RoboDK station: kr30 cnc 070119 is there hope.rdk

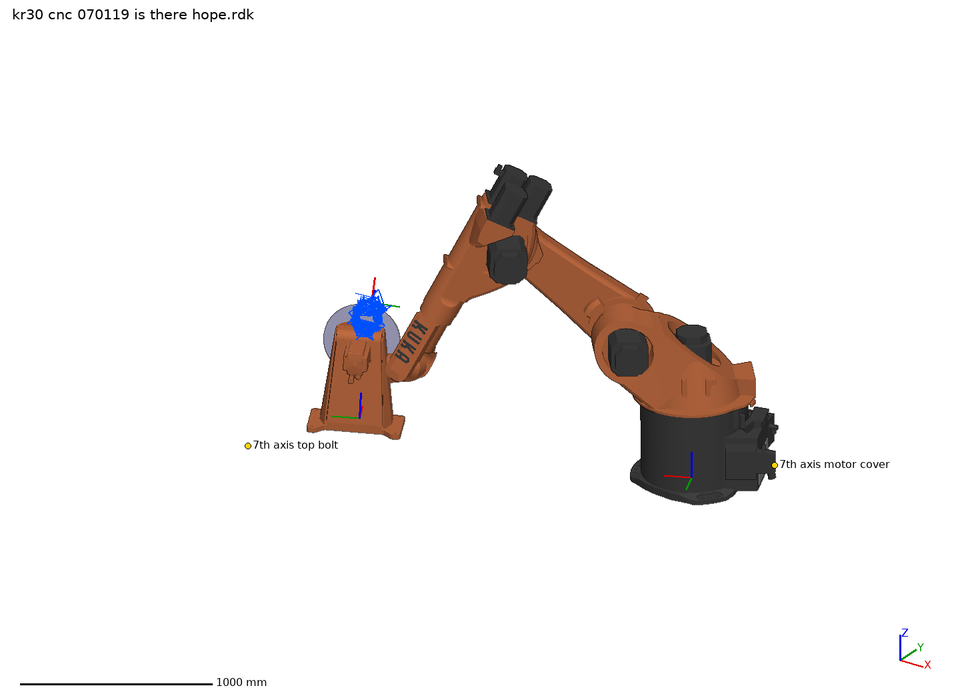
[picture v0: the station drawn from its stored meshes, robots at their saved joint values, targets as dots, program paths as lines]
Station kr30 cnc 070119 is there hope. Poses are relative to the parent item; angles as X-Y-Z fixed-axis rotations.
  - frame KUKA KR 30 HA Base at (1535.48, 628.29, -1072.61) mm, rotated rx 0 ry 0 rz -156.31 deg
    - robot KUKA KR 30 HA: 6 axes, payload 30 kg, reach 2033 mm, repeatability 0.05 mm, weight 665 kg
        modified DH rows (alpha deg, a mm, theta deg, d mm): 0, 0, 0, 815; -90, 350, 0, 0; 0, 850, -90, 0; -90, 145, 0, 820; 90, 0, 0, 0; -90, 0, 180, 170
        joint limits [-185, -135, -120, -350, -119, -350] to [185, 35, 158, 350, 119, 350]; home [0, -90, 90, 0, 0, 0]; saved at [-17.375, -41.925, 104.176, 143.001, 49.162, -26.712]
      - tool 1/2" End Mill TCP, TCP at (337.71, -2.2, 160.57) mm, rotated rx 0 ry 90 rz 0 deg, size 415.8 x 102 x 153.6 mm
    - target 7th axis top bolt (joint target) at (1966.13, 1947.63, 927.26) mm, rotated rx -179.2 ry 6.72 rz -171.11 deg; joints [-17.018, -71.525, 110.046, 168.711, 45.865, -170.331, 883.939] of KUKA KR 30 HA
    - target 7th axis motor cover (joint target) at (-417, -111.35, 57.2) mm, rotated rx -135.46 ry -1.69 rz -48.75 deg; joints [-33.388, -54.543, 96.086, 147.711, 45.276, -113.831, 883.939] of KUKA KR 30 HA
  - frame KUKA KP1 MD250 Base at (172.34, -439.05, -684.5) mm, rotated rx 2 ry 0.52 rz 120.23 deg
    - robot KUKA KP1 MD250: 1 axes, payload 250 kg
        modified DH rows (alpha deg, a mm, theta deg, d mm): 0, 0, 0, 0
        base shift (70, 10, 428) mm, rotated rx 0 ry 90 rz -2 deg
        joint limits [-3600] to [3600]; home [0]; saved at [-175]
      - frame Frame 2 at (0, 0, 440) mm
  - machining project Machining Settings: C:/Users/liqui/OneDrive/Desktop/suffering.apt | rotz(5) | rotz(0)
  - program Machining (7499 instructions, listed below)
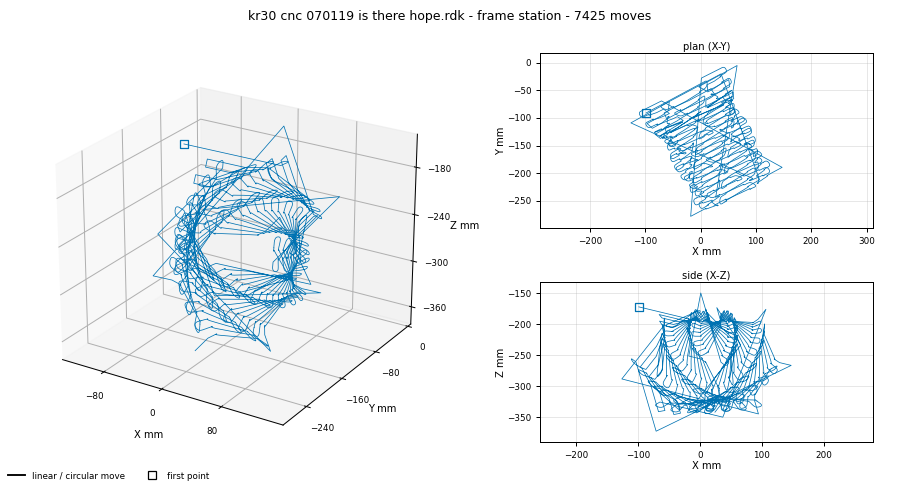
[picture p0: tool path of kr30 cnc 070119 is there hope.rdk in frame station, 7425 of 7425 moves have a stored position in this frame; points joined in program order, loops and branches not executed]

--- program Machining (robot KUKA KR 30 HA) ---
  Smooth(1)
  Set Ref.: Frame 2
  Set Tool: 1/2" End Mill TCP
  Show 1/2" End Mill TCP
  Print: /'1001'
  Print: /''
  Print: /'Flow1'
  Set speed (1000.0 mm/s)
  Set speed (1000.0 mm/s)
  MoveJ 1 to (79.06, -86.72, -80.22) mm, rotated rx 42.04 ry 15.1 rz 65.25 deg; joints [-11.881, -44.556, 105.513, 149.142, 46.632, -28.661, -175]
  MoveL 2 to (79.06, -86.72, -80.22) mm, rotated rx 42.04 ry 15.1 rz 65.25 deg; joints [-11.881, -44.556, 105.513, 149.142, 46.632, -28.661, -175]
  MoveL 3 to (79.06, -86.72, -80.22) mm, rotated rx 42.04 ry 15.1 rz 65.25 deg; joints [-11.881, -44.556, 105.513, 149.142, 46.632, -28.661, -175]
  Set speed (1000.0 mm/s)
  MoveL 4 to (75.15, -42.01, -80.22) mm, rotated rx 42.04 ry 15.1 rz 65.25 deg; joints [-12.109, -45.867, 109.411, 150.046, 48.916, -30.305, -175]
  Set speed (100.0 mm/s)
  MoveL 5 to (68.81, 30.47, -80.22) mm, rotated rx 42.04 ry 15.1 rz 65.25 deg; joints [-12.508, -47.756, 115.477, 151.236, 52.637, -32.762, -175]
  MoveL 6 to (69.1, 30.91, -80.22) mm, rotated rx 42.04 ry 15.1 rz 65.25 deg; joints [-12.511, -47.788, 115.518, 151.237, 52.647, -32.767, -175]
  MoveL 7 to (69.4, 31.48, -80.12) mm, rotated rx 42.04 ry 15.1 rz 65.25 deg; joints [-12.51, -47.824, 115.571, 151.244, 52.661, -32.777, -175]
  MoveL 8 to (69.7, 31.99, -80.06) mm, rotated rx 42.04 ry 15.1 rz 65.25 deg; joints [-12.511, -47.858, 115.619, 151.248, 52.674, -32.786, -175]
  MoveL 9 to (70, 32.47, -80.04) mm, rotated rx 42.04 ry 15.1 rz 65.25 deg; joints [-12.513, -47.891, 115.664, 151.25, 52.685, -32.792, -175]
  MoveL 10 to (72, 35.54, -80.04) mm, rotated rx 42.04 ry 15.1 rz 65.25 deg; joints [-12.532, -48.109, 115.952, 151.254, 52.75, -32.827, -175]
  MoveL 11 to (72.84, 36.72, -80.13) mm, rotated rx 42.04 ry 15.1 rz 65.25 deg; joints [-12.542, -48.197, 116.063, 151.249, 52.771, -32.836, -175]
  MoveL 12 to (73.64, 37.61, -80.4) mm, rotated rx 42.04 ry 15.1 rz 65.25 deg; joints [-12.559, -48.272, 116.146, 151.233, 52.781, -32.834, -175]
  MoveL 13 to (74.38, 38.19, -80.84) mm, rotated rx 42.04 ry 15.1 rz 65.25 deg; joints [-12.581, -48.334, 116.201, 151.204, 52.779, -32.82, -175]
  MoveL 14 to (74.73, 38.37, -81.13) mm, rotated rx 42.04 ry 15.1 rz 65.25 deg; joints [-12.594, -48.361, 116.218, 151.185, 52.774, -32.809, -175]
  MoveL 15 to (75.07, 38.48, -81.46) mm, rotated rx 42.04 ry 15.1 rz 65.25 deg; joints [-12.609, -48.384, 116.229, 151.163, 52.765, -32.795, -175]
  MoveL 16 to (75.72, 38.47, -82.26) mm, rotated rx 42.04 ry 15.1 rz 65.25 deg; joints [-12.642, -48.421, 116.229, 151.11, 52.739, -32.759, -175]
  MoveL 17 to (76.31, 38.17, -83.24) mm, rotated rx 42.04 ry 15.1 rz 65.25 deg; joints [-12.682, -48.445, 116.202, 151.045, 52.701, -32.712, -175]
  MoveL 18 to (77.36, 36.66, -85.72) mm, rotated rx 42.04 ry 15.1 rz 65.25 deg; joints [-12.777, -48.455, 116.064, 150.878, 52.589, -32.582, -175]
  MoveL 19 to (77.93, 34.52, -88.21) mm, rotated rx 42.04 ry 15.1 rz 65.25 deg; joints [-12.867, -48.415, 115.865, 150.712, 52.467, -32.446, -175]
  MoveL 20 to (77.76, 32.29, -89.98) mm, rotated rx 42.04 ry 15.1 rz 65.25 deg; joints [-12.927, -48.329, 115.655, 150.594, 52.371, -32.344, -175]
  MoveL 21 to (77.39, 31.15, -90.6) mm, rotated rx 42.04 ry 15.1 rz 65.25 deg; joints [-12.946, -48.269, 115.547, 150.554, 52.332, -32.306, -175]
  MoveL 22 to (76.84, 29.98, -91.05) mm, rotated rx 42.04 ry 15.1 rz 65.25 deg; joints [-12.957, -48.197, 115.435, 150.526, 52.3, -32.277, -175]
  MoveL 23 to (75.19, 27.58, -91.4) mm, rotated rx 42.04 ry 15.1 rz 65.25 deg; joints [-12.956, -48.019, 115.205, 150.507, 52.254, -32.244, -175]
  MoveL 24 to (73.18, 25.16, -91.41) mm, rotated rx 42.04 ry 15.1 rz 65.25 deg; joints [-12.941, -47.82, 114.97, 150.511, 52.22, -32.229, -175]
  MoveL 25 to (72.87, 24.77, -91.43) mm, rotated rx 42.04 ry 15.1 rz 65.25 deg; joints [-12.94, -47.789, 114.933, 150.51, 52.214, -32.225, -175]
  MoveL 26 to (72.6, 24.4, -91.47) mm, rotated rx 42.04 ry 15.1 rz 65.25 deg; joints [-12.939, -47.761, 114.897, 150.508, 52.208, -32.221, -175]
  MoveL 27 to (72.37, 24.06, -91.53) mm, rotated rx 42.04 ry 15.1 rz 65.25 deg; joints [-12.939, -47.735, 114.864, 150.505, 52.201, -32.216, -175]
  MoveL 28 to (72.11, 23.7, -91.58) mm, rotated rx 42.04 ry 15.1 rz 65.25 deg; joints [-12.939, -47.708, 114.829, 150.502, 52.194, -32.211, -175]
  MoveL 29 to (71.77, 23.27, -91.6) mm, rotated rx 42.04 ry 15.1 rz 65.25 deg; joints [-12.937, -47.674, 114.787, 150.501, 52.187, -32.207, -175]
  MoveL 30 to (71.37, 22.75, -91.64) mm, rotated rx 42.04 ry 15.1 rz 65.25 deg; joints [-12.936, -47.633, 114.737, 150.5, 52.179, -32.202, -175]
  MoveL 31 to (71.04, 22.3, -91.7) mm, rotated rx 42.04 ry 15.1 rz 65.25 deg; joints [-12.935, -47.599, 114.693, 150.497, 52.171, -32.197, -175]
  MoveL 32 to (70.79, 21.93, -91.77) mm, rotated rx 42.04 ry 15.1 rz 65.25 deg; joints [-12.936, -47.571, 114.657, 150.493, 52.163, -32.191, -175]
  MoveL 33 to (70.54, 21.58, -91.82) mm, rotated rx 42.04 ry 15.1 rz 65.25 deg; joints [-12.936, -47.545, 114.623, 150.49, 52.157, -32.186, -175]
  MoveL 34 to (70.24, 21.2, -91.84) mm, rotated rx 42.04 ry 15.1 rz 65.25 deg; joints [-12.934, -47.515, 114.586, 150.489, 52.151, -32.183, -175]
  MoveL 35 to (69.91, 20.8, -91.84) mm, rotated rx 42.04 ry 15.1 rz 65.25 deg; joints [-12.932, -47.482, 114.547, 150.49, 52.145, -32.18, -175]
  MoveL 36 to (69.56, 20.38, -91.85) mm, rotated rx 42.04 ry 15.1 rz 65.25 deg; joints [-12.929, -47.448, 114.506, 150.491, 52.139, -32.177, -175]
  MoveL 37 to (69.21, 19.93, -91.86) mm, rotated rx 42.04 ry 15.1 rz 65.25 deg; joints [-12.927, -47.412, 114.463, 150.49, 52.131, -32.173, -175]
  MoveL 38 to (68.81, 19.4, -91.89) mm, rotated rx 42.04 ry 15.1 rz 65.25 deg; joints [-12.925, -47.371, 114.412, 150.489, 52.122, -32.168, -175]
  MoveL 39 to (68.49, 18.91, -91.96) mm, rotated rx 42.04 ry 15.1 rz 65.25 deg; joints [-12.924, -47.335, 114.364, 150.485, 52.112, -32.16, -175]
  MoveL 40 to (68.26, 18.52, -92.06) mm, rotated rx 42.04 ry 15.1 rz 65.25 deg; joints [-12.926, -47.309, 114.326, 150.478, 52.102, -32.153, -175]
  MoveL 41 to (68.25, 18.52, -92.3) mm, rotated rx 42.04 ry 15.1 rz 65.25 deg; joints [-12.936, -47.307, 114.324, 150.466, 52.103, -32.148, -175]
  MoveL 42 to (68.39, 18.89, -92.65) mm, rotated rx 42.04 ry 15.1 rz 65.25 deg; joints [-12.953, -47.325, 114.353, 150.45, 52.115, -32.147, -175]
  MoveL 43 to (69.21, 19.13, -93.61) mm, rotated rx 42.04 ry 15.1 rz 65.25 deg; joints [-12.994, -47.379, 114.374, 150.389, 52.095, -32.109, -175]
  MoveL 44 to (68.99, 17.01, -93.61) mm, rotated rx 42.04 ry 15.1 rz 65.25 deg; joints [-12.981, -47.301, 114.192, 150.365, 52.003, -32.05, -175]
  MoveL 45 to (68.79, 14.72, -93.74) mm, rotated rx 42.04 ry 15.1 rz 65.25 deg; joints [-12.972, -47.219, 113.996, 150.33, 51.902, -31.982, -175]
  MoveL 46 to (68.58, 12.55, -93.8) mm, rotated rx 42.04 ry 15.1 rz 65.25 deg; joints [-12.961, -47.139, 113.809, 150.302, 51.807, -31.919, -175]
  MoveL 47 to (68.38, 10.44, -93.93) mm, rotated rx 42.04 ry 15.1 rz 65.25 deg; joints [-12.954, -47.062, 113.627, 150.27, 51.714, -31.856, -175]
  MoveL 48 to (68.18, 8.3, -94.09) mm, rotated rx 42.04 ry 15.1 rz 65.25 deg; joints [-12.947, -46.984, 113.442, 150.236, 51.62, -31.791, -175]
  MoveL 49 to (67.98, 6.19, -94.21) mm, rotated rx 42.04 ry 15.1 rz 65.25 deg; joints [-12.94, -46.906, 113.259, 150.203, 51.527, -31.728, -175]
  MoveL 50 to (67.78, 4.06, -94.42) mm, rotated rx 42.04 ry 15.1 rz 65.25 deg; joints [-12.935, -46.827, 113.073, 150.166, 51.433, -31.662, -175]
  MoveL 51 to (67.57, 1.94, -94.54) mm, rotated rx 42.04 ry 15.1 rz 65.25 deg; joints [-12.927, -46.748, 112.889, 150.134, 51.34, -31.599, -175]
  MoveL 52 to (67.36, -0.19, -94.59) mm, rotated rx 42.04 ry 15.1 rz 65.25 deg; joints [-12.917, -46.669, 112.704, 150.105, 51.247, -31.536, -175]
  MoveL 53 to (67.14, -2.34, -94.74) mm, rotated rx 42.04 ry 15.1 rz 65.25 deg; joints [-12.91, -46.588, 112.517, 150.07, 51.153, -31.471, -175]
  MoveL 54 to (66.92, -4.55, -94.92) mm, rotated rx 42.04 ry 15.1 rz 65.25 deg; joints [-12.904, -46.505, 112.323, 150.033, 51.056, -31.403, -175]
  MoveL 55 to (66.69, -6.77, -95.1) mm, rotated rx 42.04 ry 15.1 rz 65.25 deg; joints [-12.898, -46.421, 112.128, 149.995, 50.959, -31.335, -175]
  MoveL 56 to (66.49, -8.63, -95.34) mm, rotated rx 42.04 ry 15.1 rz 65.25 deg; joints [-12.896, -46.349, 111.963, 149.959, 50.878, -31.275, -175]
  MoveL 57 to (66.21, -11.29, -95.45) mm, rotated rx 42.04 ry 15.1 rz 65.25 deg; joints [-12.885, -46.248, 111.731, 149.919, 50.762, -31.196, -175]
  Set speed (1000.0 mm/s)
  MoveL 58 to (70.16, -56.42, -95.45) mm, rotated rx 42.04 ry 15.1 rz 65.25 deg; joints [-12.627, -45.013, 107.885, 149.106, 48.456, -29.584, -175]
  Set speed (1000.0 mm/s)
  MoveL 59 to (64.44, -56.92, -107.33) mm, rotated rx 42.04 ry 15.1 rz 65.25 deg; joints [-13.086, -44.596, 107.594, 148.598, 48.671, -29.432, -175]
  Set speed (100.0 mm/s)
  MoveL 60 to (61.94, -28.34, -107.33) mm, rotated rx 42.04 ry 15.1 rz 65.25 deg; joints [-13.255, -45.385, 110.042, 149.126, 50.129, -30.478, -175]
  MoveL 61 to (62.35, -26.67, -107.08) mm, rotated rx 42.04 ry 15.1 rz 65.25 deg; joints [-13.256, -45.465, 110.196, 149.157, 50.193, -30.527, -175]
  MoveL 62 to (62.8, -24.7, -107.02) mm, rotated rx 42.04 ry 15.1 rz 65.25 deg; joints [-13.266, -45.555, 110.375, 149.183, 50.271, -30.581, -175]
  MoveL 63 to (63.26, -22.7, -106.87) mm, rotated rx 42.04 ry 15.1 rz 65.25 deg; joints [-13.272, -45.648, 110.556, 149.213, 50.349, -30.637, -175]
  MoveL 64 to (63.83, -20.3, -106.74) mm, rotated rx 42.04 ry 15.1 rz 65.25 deg; joints [-13.282, -45.759, 110.773, 149.246, 50.442, -30.703, -175]
  MoveL 65 to (64.3, -18.22, -106.74) mm, rotated rx 42.04 ry 15.1 rz 65.25 deg; joints [-13.295, -45.854, 110.96, 149.269, 50.524, -30.758, -175]
  MoveL 66 to (64.81, -15.92, -106.58) mm, rotated rx 42.04 ry 15.1 rz 65.25 deg; joints [-13.303, -45.959, 111.167, 149.303, 50.614, -30.822, -175]
  MoveL 67 to (65.26, -13.98, -106.39) mm, rotated rx 42.04 ry 15.1 rz 65.25 deg; joints [-13.307, -46.048, 111.343, 149.333, 50.689, -30.877, -175]
  MoveL 68 to (65.72, -11.98, -106.3) mm, rotated rx 42.04 ry 15.1 rz 65.25 deg; joints [-13.316, -46.139, 111.523, 149.359, 50.767, -30.931, -175]
  MoveL 69 to (66.18, -9.9, -106.08) mm, rotated rx 42.04 ry 15.1 rz 65.25 deg; joints [-13.321, -46.234, 111.711, 149.393, 50.848, -30.99, -175]
  MoveL 70 to (66.64, -7.83, -105.93) mm, rotated rx 42.04 ry 15.1 rz 65.25 deg; joints [-13.327, -46.328, 111.896, 149.423, 50.928, -31.047, -175]
  MoveL 71 to (67.1, -5.77, -105.82) mm, rotated rx 42.04 ry 15.1 rz 65.25 deg; joints [-13.336, -46.421, 112.081, 149.45, 51.009, -31.103, -175]
  MoveL 72 to (67.55, -3.68, -105.65) mm, rotated rx 42.04 ry 15.1 rz 65.25 deg; joints [-13.342, -46.515, 112.268, 149.481, 51.091, -31.161, -175]
  MoveL 73 to (68, -1.6, -105.51) mm, rotated rx 42.04 ry 15.1 rz 65.25 deg; joints [-13.35, -46.608, 112.454, 149.51, 51.172, -31.218, -175]
  MoveL 74 to (68.47, 0.52, -105.44) mm, rotated rx 42.04 ry 15.1 rz 65.25 deg; joints [-13.361, -46.703, 112.642, 149.535, 51.255, -31.274, -175]
  MoveL 75 to (68.91, 2.61, -105.23) mm, rotated rx 42.04 ry 15.1 rz 65.25 deg; joints [-13.365, -46.796, 112.829, 149.567, 51.337, -31.333, -175]
  MoveL 76 to (69.35, 4.68, -105.11) mm, rotated rx 42.04 ry 15.1 rz 65.25 deg; joints [-13.374, -46.888, 113.013, 149.595, 51.418, -31.389, -175]
  MoveL 77 to (69.81, 6.8, -104.99) mm, rotated rx 42.04 ry 15.1 rz 65.25 deg; joints [-13.382, -46.982, 113.201, 149.622, 51.5, -31.446, -175]
  MoveL 78 to (70.05, 8.56, -104.78) mm, rotated rx 42.04 ry 15.1 rz 65.25 deg; joints [-13.385, -47.052, 113.356, 149.653, 51.574, -31.499, -175]
  MoveL 79 to (70.11, 10.03, -104.43) mm, rotated rx 42.04 ry 15.1 rz 65.25 deg; joints [-13.38, -47.103, 113.485, 149.691, 51.641, -31.552, -175]
  MoveL 80 to (69.98, 11.23, -103.9) mm, rotated rx 42.04 ry 15.1 rz 65.25 deg; joints [-13.366, -47.134, 113.591, 149.737, 51.702, -31.606, -175]
  MoveL 81 to (69.2, 9.9, -103.04) mm, rotated rx 42.04 ry 15.1 rz 65.25 deg; joints [-13.322, -47.05, 113.478, 149.777, 51.668, -31.607, -175]
  MoveL 82 to (69.54, 10.63, -103.04) mm, rotated rx 42.04 ry 15.1 rz 65.25 deg; joints [-13.327, -47.093, 113.544, 149.781, 51.69, -31.62, -175]
  MoveL 83 to (69.9, 11.23, -103.04) mm, rotated rx 42.04 ry 15.1 rz 65.25 deg; joints [-13.331, -47.134, 113.601, 149.783, 51.705, -31.628, -175]
  MoveL 84 to (70.3, 11.73, -103.04) mm, rotated rx 42.04 ry 15.1 rz 65.25 deg; joints [-13.334, -47.174, 113.649, 149.782, 51.712, -31.632, -175]
  MoveL 85 to (70.75, 12.22, -103.02) mm, rotated rx 42.04 ry 15.1 rz 65.25 deg; joints [-13.337, -47.217, 113.699, 149.782, 51.718, -31.635, -175]
  MoveL 86 to (71.28, 12.77, -102.98) mm, rotated rx 42.04 ry 15.1 rz 65.25 deg; joints [-13.339, -47.267, 113.754, 149.781, 51.723, -31.637, -175]
  MoveL 87 to (72.8, 14.21, -102.98) mm, rotated rx 42.04 ry 15.1 rz 65.25 deg; joints [-13.348, -47.405, 113.899, 149.773, 51.731, -31.638, -175]
  MoveL 88 to (73.12, 14.53, -102.96) mm, rotated rx 42.04 ry 15.1 rz 65.25 deg; joints [-13.35, -47.435, 113.931, 149.772, 51.734, -31.639, -175]
  MoveL 89 to (73.88, 15.25, -102.96) mm, rotated rx 42.04 ry 15.1 rz 65.25 deg; joints [-13.355, -47.504, 114.004, 149.768, 51.738, -31.639, -175]
  MoveL 90 to (74.24, 15.6, -102.96) mm, rotated rx 42.04 ry 15.1 rz 65.25 deg; joints [-13.357, -47.537, 114.039, 149.766, 51.74, -31.639, -175]
  MoveL 91 to (74.59, 15.94, -102.94) mm, rotated rx 42.04 ry 15.1 rz 65.25 deg; joints [-13.358, -47.569, 114.074, 149.765, 51.742, -31.64, -175]
  MoveL 92 to (74.92, 16.29, -102.91) mm, rotated rx 42.04 ry 15.1 rz 65.25 deg; joints [-13.359, -47.601, 114.109, 149.765, 51.745, -31.642, -175]
  MoveL 93 to (75.21, 16.61, -102.85) mm, rotated rx 42.04 ry 15.1 rz 65.25 deg; joints [-13.359, -47.629, 114.141, 149.767, 51.749, -31.645, -175]
  MoveL 94 to (75.53, 16.95, -102.81) mm, rotated rx 42.04 ry 15.1 rz 65.25 deg; joints [-13.36, -47.66, 114.176, 149.768, 51.752, -31.647, -175]
  MoveL 95 to (75.88, 17.3, -102.79) mm, rotated rx 42.04 ry 15.1 rz 65.25 deg; joints [-13.361, -47.693, 114.211, 149.767, 51.755, -31.647, -175]
  MoveL 96 to (76.25, 17.66, -102.78) mm, rotated rx 42.04 ry 15.1 rz 65.25 deg; joints [-13.363, -47.726, 114.246, 149.765, 51.757, -31.648, -175]
  MoveL 97 to (76.6, 18.01, -102.77) mm, rotated rx 42.04 ry 15.1 rz 65.25 deg; joints [-13.365, -47.759, 114.281, 149.764, 51.759, -31.649, -175]
  MoveL 98 to (76.92, 18.35, -102.73) mm, rotated rx 42.04 ry 15.1 rz 65.25 deg; joints [-13.366, -47.79, 114.316, 149.765, 51.763, -31.651, -175]
  MoveL 99 to (77.21, 18.68, -102.67) mm, rotated rx 42.04 ry 15.1 rz 65.25 deg; joints [-13.366, -47.818, 114.349, 149.767, 51.767, -31.654, -175]
  MoveL 100 to (77.51, 19.03, -102.62) mm, rotated rx 42.04 ry 15.1 rz 65.25 deg; joints [-13.366, -47.847, 114.383, 149.768, 51.771, -31.657, -175]
  MoveL 101 to (78.5, 20.06, -102.54) mm, rotated rx 42.04 ry 15.1 rz 65.25 deg; joints [-13.369, -47.942, 114.487, 149.768, 51.78, -31.661, -175]
  MoveL 102 to (79.42, 20.81, -102.66) mm, rotated rx 42.04 ry 15.1 rz 65.25 deg; joints [-13.38, -48.021, 114.562, 149.754, 51.778, -31.654, -175]
  MoveL 103 to (80.25, 21.25, -103) mm, rotated rx 42.04 ry 15.1 rz 65.25 deg; joints [-13.397, -48.084, 114.607, 149.727, 51.766, -31.635, -175]
  MoveL 104 to (80.64, 21.36, -103.25) mm, rotated rx 42.04 ry 15.1 rz 65.25 deg; joints [-13.408, -48.111, 114.619, 149.708, 51.756, -31.621, -175]
  MoveL 105 to (81, 21.4, -103.55) mm, rotated rx 42.04 ry 15.1 rz 65.25 deg; joints [-13.42, -48.133, 114.624, 149.686, 51.743, -31.604, -175]
  MoveL 106 to (81.67, 21.25, -104.31) mm, rotated rx 42.04 ry 15.1 rz 65.25 deg; joints [-13.451, -48.166, 114.612, 149.632, 51.71, -31.562, -175]
  MoveL 107 to (82.26, 20.8, -105.27) mm, rotated rx 42.04 ry 15.1 rz 65.25 deg; joints [-13.488, -48.183, 114.571, 149.564, 51.667, -31.508, -175]
  MoveL 108 to (83.19, 19.01, -107.84) mm, rotated rx 42.04 ry 15.1 rz 65.25 deg; joints [-13.582, -48.172, 114.401, 149.389, 51.55, -31.364, -175]
  MoveL 109 to (83.54, 16.69, -110.45) mm, rotated rx 42.04 ry 15.1 rz 65.25 deg; joints [-13.674, -48.107, 114.177, 149.214, 51.432, -31.219, -175]
  MoveL 110 to (83.4, 15.58, -111.48) mm, rotated rx 42.04 ry 15.1 rz 65.25 deg; joints [-13.708, -48.059, 114.067, 149.148, 51.387, -31.163, -175]
  MoveL 111 to (83.06, 14.5, -112.32) mm, rotated rx 42.04 ry 15.1 rz 65.25 deg; joints [-13.735, -47.999, 113.959, 149.096, 51.351, -31.12, -175]
  MoveL 112 to (82.5, 13.45, -112.97) mm, rotated rx 42.04 ry 15.1 rz 65.25 deg; joints [-13.755, -47.929, 113.854, 149.058, 51.325, -31.088, -175]
  MoveL 113 to (81.75, 12.43, -113.44) mm, rotated rx 42.04 ry 15.1 rz 65.25 deg; joints [-13.767, -47.847, 113.75, 149.035, 51.308, -31.067, -175]
  MoveL 114 to (80.78, 11.44, -113.72) mm, rotated rx 42.04 ry 15.1 rz 65.25 deg; joints [-13.771, -47.755, 113.648, 149.025, 51.3, -31.059, -175]
  MoveL 115 to (79.61, 10.48, -113.81) mm, rotated rx 42.04 ry 15.1 rz 65.25 deg; joints [-13.768, -47.652, 113.548, 149.03, 51.302, -31.062, -175]
  MoveL 116 to (77.07, 8.6, -113.81) mm, rotated rx 42.04 ry 15.1 rz 65.25 deg; joints [-13.755, -47.437, 113.35, 149.053, 51.314, -31.079, -175]
  MoveL 117 to (76.63, 8.26, -113.83) mm, rotated rx 42.04 ry 15.1 rz 65.25 deg; joints [-13.753, -47.4, 113.314, 149.056, 51.315, -31.081, -175]
  MoveL 118 to (76.14, 7.87, -113.86) mm, rotated rx 42.04 ry 15.1 rz 65.25 deg; joints [-13.752, -47.358, 113.273, 149.058, 51.316, -31.083, -175]
  MoveL 119 to (75.57, 7.38, -113.96) mm, rotated rx 42.04 ry 15.1 rz 65.25 deg; joints [-13.752, -47.306, 113.221, 149.057, 51.315, -31.082, -175]
  MoveL 120 to (75.09, 6.99, -113.99) mm, rotated rx 42.04 ry 15.1 rz 65.25 deg; joints [-13.751, -47.264, 113.18, 149.059, 51.316, -31.083, -175]
  MoveL 121 to (74.65, 6.66, -114.01) mm, rotated rx 42.04 ry 15.1 rz 65.25 deg; joints [-13.749, -47.227, 113.145, 149.062, 51.317, -31.085, -175]
  MoveL 122 to (74.25, 6.35, -114.02) mm, rotated rx 42.04 ry 15.1 rz 65.25 deg; joints [-13.747, -47.193, 113.112, 149.065, 51.318, -31.087, -175]
  MoveL 123 to (73.89, 6.07, -114.03) mm, rotated rx 42.04 ry 15.1 rz 65.25 deg; joints [-13.746, -47.162, 113.082, 149.067, 51.319, -31.089, -175]
  MoveL 124 to (72.24, 4.84, -114.04) mm, rotated rx 42.04 ry 15.1 rz 65.25 deg; joints [-13.738, -47.022, 112.952, 149.081, 51.325, -31.099, -175]
  MoveL 125 to (71.84, 4.52, -114.08) mm, rotated rx 42.04 ry 15.1 rz 65.25 deg; joints [-13.737, -46.987, 112.918, 149.082, 51.326, -31.099, -175]
  MoveL 126 to (71.48, 4.21, -114.13) mm, rotated rx 42.04 ry 15.1 rz 65.25 deg; joints [-13.737, -46.955, 112.885, 149.082, 51.325, -31.099, -175]
  MoveL 127 to (71.15, 3.89, -114.2) mm, rotated rx 42.04 ry 15.1 rz 65.25 deg; joints [-13.738, -46.925, 112.852, 149.08, 51.323, -31.097, -175]
  MoveL 128 to (70.81, 3.54, -114.26) mm, rotated rx 42.04 ry 15.1 rz 65.25 deg; joints [-13.738, -46.892, 112.816, 149.079, 51.32, -31.095, -175]
  MoveL 129 to (70.44, 3.13, -114.29) mm, rotated rx 42.04 ry 15.1 rz 65.25 deg; joints [-13.736, -46.857, 112.775, 149.078, 51.315, -31.092, -175]
  MoveL 130 to (70.06, 2.58, -114.3) mm, rotated rx 42.04 ry 15.1 rz 65.25 deg; joints [-13.733, -46.816, 112.722, 149.077, 51.304, -31.085, -175]
  MoveL 131 to (69.68, 1.9, -114.3) mm, rotated rx 42.04 ry 15.1 rz 65.25 deg; joints [-13.728, -46.772, 112.659, 149.075, 51.286, -31.074, -175]
  MoveL 132 to (71.32, 2.95, -115.86) mm, rotated rx 42.04 ry 15.1 rz 65.25 deg; joints [-13.798, -46.896, 112.752, 148.978, 51.275, -31.023, -175]
  MoveL 133 to (70.55, 0.71, -115.99) mm, rotated rx 42.04 ry 15.1 rz 65.25 deg; joints [-13.789, -46.779, 112.549, 148.954, 51.199, -30.97, -175]
  MoveL 134 to (69.81, -1.4, -116.1) mm, rotated rx 42.04 ry 15.1 rz 65.25 deg; joints [-13.779, -46.667, 112.356, 148.932, 51.128, -30.921, -175]
  MoveL 135 to (69.12, -3.44, -116.26) mm, rotated rx 42.04 ry 15.1 rz 65.25 deg; joints [-13.772, -46.56, 112.17, 148.907, 51.058, -30.871, -175]
  MoveL 136 to (68.42, -5.46, -116.37) mm, rotated rx 42.04 ry 15.1 rz 65.25 deg; joints [-13.763, -46.453, 111.985, 148.886, 50.99, -30.824, -175]
  MoveL 137 to (67.72, -7.47, -116.48) mm, rotated rx 42.04 ry 15.1 rz 65.25 deg; joints [-13.754, -46.347, 111.801, 148.864, 50.921, -30.776, -175]
  MoveL 138 to (67.03, -9.5, -116.7) mm, rotated rx 42.04 ry 15.1 rz 65.25 deg; joints [-13.749, -46.24, 111.614, 148.836, 50.852, -30.725, -175]
  MoveL 139 to (66.33, -11.51, -116.92) mm, rotated rx 42.04 ry 15.1 rz 65.25 deg; joints [-13.745, -46.133, 111.427, 148.808, 50.783, -30.674, -175]
  MoveL 140 to (65.62, -13.53, -117.04) mm, rotated rx 42.04 ry 15.1 rz 65.25 deg; joints [-13.736, -46.025, 111.242, 148.785, 50.714, -30.626, -175]
  MoveL 141 to (64.9, -15.54, -117.04) mm, rotated rx 42.04 ry 15.1 rz 65.25 deg; joints [-13.723, -45.918, 111.059, 148.769, 50.646, -30.581, -175]
  MoveL 142 to (64.19, -17.55, -117.15) mm, rotated rx 42.04 ry 15.1 rz 65.25 deg; joints [-13.714, -45.81, 110.873, 148.746, 50.577, -30.533, -175]
  MoveL 143 to (63.46, -19.59, -117.35) mm, rotated rx 42.04 ry 15.1 rz 65.25 deg; joints [-13.709, -45.701, 110.683, 148.718, 50.508, -30.481, -175]
  MoveL 144 to (62.79, -21.48, -117.53) mm, rotated rx 42.04 ry 15.1 rz 65.25 deg; joints [-13.703, -45.598, 110.507, 148.693, 50.443, -30.434, -175]
  MoveL 145 to (62.16, -23.23, -117.75) mm, rotated rx 42.04 ry 15.1 rz 65.25 deg; joints [-13.701, -45.504, 110.343, 148.666, 50.384, -30.389, -175]
  MoveL 146 to (61.5, -25.08, -117.84) mm, rotated rx 42.04 ry 15.1 rz 65.25 deg; joints [-13.692, -45.404, 110.171, 148.646, 50.32, -30.344, -175]
  MoveL 147 to (60.79, -27.05, -117.85) mm, rotated rx 42.04 ry 15.1 rz 65.25 deg; joints [-13.68, -45.299, 109.99, 148.628, 50.252, -30.298, -175]
  MoveL 148 to (59.86, -29.6, -117.95) mm, rotated rx 42.04 ry 15.1 rz 65.25 deg; joints [-13.667, -45.161, 109.753, 148.6, 50.165, -30.237, -175]
  MoveL 149 to (59.16, -31.51, -118.16) mm, rotated rx 42.04 ry 15.1 rz 65.25 deg; joints [-13.663, -45.056, 109.573, 148.572, 50.1, -30.188, -175]
  MoveL 150 to (58.39, -33.57, -118.36) mm, rotated rx 42.04 ry 15.1 rz 65.25 deg; joints [-13.658, -44.942, 109.379, 148.544, 50.03, -30.136, -175]
  MoveL 151 to (57.67, -35.46, -118.65) mm, rotated rx 42.04 ry 15.1 rz 65.25 deg; joints [-13.657, -44.837, 109.199, 148.512, 49.967, -30.086, -175]
  MoveL 152 to (56.99, -37.32, -118.78) mm, rotated rx 42.04 ry 15.1 rz 65.25 deg; joints [-13.65, -44.735, 109.024, 148.488, 49.903, -30.039, -175]
  MoveL 153 to (56.28, -39.29, -118.79) mm, rotated rx 42.04 ry 15.1 rz 65.25 deg; joints [-13.638, -44.629, 108.84, 148.469, 49.834, -29.992, -175]
  MoveL 154 to (55.63, -40.94, -119.02) mm, rotated rx 42.04 ry 15.1 rz 65.25 deg; joints [-13.636, -44.535, 108.682, 148.442, 49.779, -29.949, -175]
  Set speed (1000.0 mm/s)
  MoveL 155 to (57.9, -66.9, -119.02) mm, rotated rx 42.04 ry 15.1 rz 65.25 deg; joints [-13.477, -43.809, 106.442, 147.946, 48.454, -28.973, -175]
  Set speed (1000.0 mm/s)
  MoveL 156 to (51.39, -67.47, -130.21) mm, rotated rx 42.04 ry 15.1 rz 65.25 deg; joints [-13.901, -43.342, 106.117, 147.491, 48.679, -28.855, -175]
  Set speed (100.0 mm/s)
  MoveL 157 to (49.64, -47.38, -130.21) mm, rotated rx 42.04 ry 15.1 rz 65.25 deg; joints [-14.03, -43.903, 107.855, 147.878, 49.704, -29.622, -175]
  MoveL 158 to (50.6, -45.47, -130.21) mm, rotated rx 42.04 ry 15.1 rz 65.25 deg; joints [-14.042, -44.022, 108.038, 147.891, 49.761, -29.661, -175]
  MoveL 159 to (51.63, -43.49, -130.11) mm, rotated rx 42.04 ry 15.1 rz 65.25 deg; joints [-14.052, -44.148, 108.23, 147.909, 49.819, -29.702, -175]
  MoveL 160 to (52.75, -41.43, -129.82) mm, rotated rx 42.04 ry 15.1 rz 65.25 deg; joints [-14.054, -44.283, 108.434, 147.937, 49.878, -29.748, -175]
  MoveL 161 to (53.82, -39.45, -129.47) mm, rotated rx 42.04 ry 15.1 rz 65.25 deg; joints [-14.054, -44.414, 108.63, 147.966, 49.933, -29.794, -175]
  MoveL 162 to (54.78, -37.62, -129.28) mm, rotated rx 42.04 ry 15.1 rz 65.25 deg; joints [-14.059, -44.531, 108.808, 147.987, 49.986, -29.834, -175]
  MoveL 163 to (55.67, -35.88, -129.15) mm, rotated rx 42.04 ry 15.1 rz 65.25 deg; joints [-14.066, -44.642, 108.976, 148.005, 50.036, -29.871, -175]
  MoveL 164 to (56.61, -34.06, -129.1) mm, rotated rx 42.04 ry 15.1 rz 65.25 deg; joints [-14.076, -44.757, 109.151, 148.019, 50.09, -29.907, -175]
  MoveL 165 to (57.57, -32.15, -129.07) mm, rotated rx 42.04 ry 15.1 rz 65.25 deg; joints [-14.088, -44.876, 109.333, 148.032, 50.146, -29.944, -175]
  MoveL 166 to (58.53, -30.26, -128.96) mm, rotated rx 42.04 ry 15.1 rz 65.25 deg; joints [-14.096, -44.995, 109.515, 148.05, 50.2, -29.983, -175]
  MoveL 167 to (59.58, -28.22, -128.7) mm, rotated rx 42.04 ry 15.1 rz 65.25 deg; joints [-14.1, -45.124, 109.712, 148.075, 50.259, -30.028, -175]
  MoveL 168 to (60.66, -26.08, -128.51) mm, rotated rx 42.04 ry 15.1 rz 65.25 deg; joints [-14.108, -45.259, 109.918, 148.097, 50.321, -30.074, -175]
  MoveL 169 to (61.71, -24, -128.31) mm, rotated rx 42.04 ry 15.1 rz 65.25 deg; joints [-14.114, -45.39, 110.118, 148.12, 50.381, -30.118, -175]
  MoveL 170 to (62.67, -22.09, -128.2) mm, rotated rx 42.04 ry 15.1 rz 65.25 deg; joints [-14.123, -45.509, 110.299, 148.137, 50.436, -30.157, -175]
  MoveL 171 to (64.55, -18.31, -127.92) mm, rotated rx 42.04 ry 15.1 rz 65.25 deg; joints [-14.138, -45.745, 110.659, 148.172, 50.544, -30.234, -175]
  MoveL 172 to (65.53, -16.37, -127.86) mm, rotated rx 42.04 ry 15.1 rz 65.25 deg; joints [-14.149, -45.867, 110.843, 148.186, 50.6, -30.272, -175]
  MoveL 173 to (66.47, -14.45, -127.64) mm, rotated rx 42.04 ry 15.1 rz 65.25 deg; joints [-14.153, -45.986, 111.025, 148.209, 50.655, -30.313, -175]
  MoveL 174 to (67.4, -12.56, -127.48) mm, rotated rx 42.04 ry 15.1 rz 65.25 deg; joints [-14.16, -46.103, 111.205, 148.227, 50.709, -30.352, -175]
  MoveL 175 to (68.32, -10.66, -127.29) mm, rotated rx 42.04 ry 15.1 rz 65.25 deg; joints [-14.166, -46.22, 111.385, 148.247, 50.764, -30.392, -175]
  MoveL 176 to (69.29, -8.71, -127.2) mm, rotated rx 42.04 ry 15.1 rz 65.25 deg; joints [-14.176, -46.341, 111.568, 148.262, 50.819, -30.43, -175]
  MoveL 177 to (70.28, -6.66, -127.07) mm, rotated rx 42.04 ry 15.1 rz 65.25 deg; joints [-14.185, -46.467, 111.76, 148.279, 50.878, -30.471, -175]
  MoveL 178 to (71.14, -4.97, -127.01) mm, rotated rx 42.04 ry 15.1 rz 65.25 deg; joints [-14.195, -46.573, 111.919, 148.29, 50.924, -30.502, -175]
  MoveL 179 to (70.55, -4.67, -126.13) mm, rotated rx 42.04 ry 15.1 rz 65.25 deg; joints [-14.161, -46.552, 111.948, 148.352, 50.96, -30.551, -175]
  MoveL 180 to (70.23, -4.83, -125.71) mm, rotated rx 42.04 ry 15.1 rz 65.25 deg; joints [-14.143, -46.529, 111.935, 148.377, 50.964, -30.566, -175]
  MoveL 181 to (70.16, -4.82, -125.44) mm, rotated rx 42.04 ry 15.1 rz 65.25 deg; joints [-14.132, -46.527, 111.939, 148.393, 50.967, -30.575, -175]
  MoveL 182 to (70.42, -4.62, -125.32) mm, rotated rx 42.04 ry 15.1 rz 65.25 deg; joints [-14.129, -46.55, 111.962, 148.397, 50.966, -30.577, -175]
  MoveL 183 to (70.79, -4.36, -125.26) mm, rotated rx 42.04 ry 15.1 rz 65.25 deg; joints [-14.128, -46.581, 111.99, 148.397, 50.964, -30.575, -175]
  MoveL 184 to (71.27, -4.07, -125.23) mm, rotated rx 42.04 ry 15.1 rz 65.25 deg; joints [-14.129, -46.62, 112.024, 148.393, 50.959, -30.571, -175]
  MoveL 185 to (71.86, -3.7, -125.19) mm, rotated rx 42.04 ry 15.1 rz 65.25 deg; joints [-14.13, -46.668, 112.065, 148.389, 50.954, -30.566, -175]
  MoveL 186 to (72.41, -3.38, -125.16) mm, rotated rx 42.04 ry 15.1 rz 65.25 deg; joints [-14.132, -46.711, 112.101, 148.384, 50.948, -30.56, -175]
  MoveL 187 to (72.86, -3.13, -125.16) mm, rotated rx 42.04 ry 15.1 rz 65.25 deg; joints [-14.133, -46.747, 112.13, 148.379, 50.943, -30.555, -175]
  MoveL 188 to (73.28, -2.88, -125.15) mm, rotated rx 42.04 ry 15.1 rz 65.25 deg; joints [-14.135, -46.781, 112.158, 148.375, 50.938, -30.551, -175]
  MoveL 189 to (74.16, -2.32, -125.07) mm, rotated rx 42.04 ry 15.1 rz 65.25 deg; joints [-14.136, -46.852, 112.221, 148.37, 50.93, -30.544, -175]
  MoveL 190 to (74.63, -2.02, -125.02) mm, rotated rx 42.04 ry 15.1 rz 65.25 deg; joints [-14.136, -46.891, 112.254, 148.368, 50.927, -30.541, -175]
  MoveL 191 to (75.05, -1.73, -124.95) mm, rotated rx 42.04 ry 15.1 rz 65.25 deg; joints [-14.135, -46.926, 112.287, 148.367, 50.924, -30.539, -175]
  MoveL 192 to (75.43, -1.46, -124.88) mm, rotated rx 42.04 ry 15.1 rz 65.25 deg; joints [-14.134, -46.958, 112.317, 148.368, 50.922, -30.538, -175]
  MoveL 193 to (75.82, -1.2, -124.82) mm, rotated rx 42.04 ry 15.1 rz 65.25 deg; joints [-14.134, -46.99, 112.346, 148.367, 50.919, -30.536, -175]
  MoveL 194 to (76.23, -0.94, -124.79) mm, rotated rx 42.04 ry 15.1 rz 65.25 deg; joints [-14.135, -47.023, 112.374, 148.364, 50.915, -30.533, -175]
  MoveL 195 to (76.68, -0.68, -124.77) mm, rotated rx 42.04 ry 15.1 rz 65.25 deg; joints [-14.136, -47.059, 112.404, 148.36, 50.911, -30.528, -175]
  MoveL 196 to (79.87, 1.12, -124.77) mm, rotated rx 42.04 ry 15.1 rz 65.25 deg; joints [-14.149, -47.311, 112.606, 148.323, 50.871, -30.488, -175]
  MoveL 197 to (81.34, 1.82, -124.79) mm, rotated rx 42.04 ry 15.1 rz 65.25 deg; joints [-14.156, -47.423, 112.688, 148.302, 50.847, -30.465, -175]
  MoveL 198 to (81.89, 1.98, -124.81) mm, rotated rx 42.04 ry 15.1 rz 65.25 deg; joints [-14.158, -47.462, 112.71, 148.292, 50.833, -30.452, -175]
  MoveL 199 to (82.33, 2.03, -124.85) mm, rotated rx 42.04 ry 15.1 rz 65.25 deg; joints [-14.16, -47.49, 112.72, 148.282, 50.818, -30.439, -175]
  MoveL 200 to (82.67, 1.97, -124.89) mm, rotated rx 42.04 ry 15.1 rz 65.25 deg; joints [-14.161, -47.509, 112.72, 148.272, 50.802, -30.426, -175]
  MoveL 201 to (82.8, 1.91, -124.92) mm, rotated rx 42.04 ry 15.1 rz 65.25 deg; joints [-14.162, -47.515, 112.716, 148.268, 50.794, -30.419, -175]
  MoveL 202 to (82.91, 1.82, -124.94) mm, rotated rx 42.04 ry 15.1 rz 65.25 deg; joints [-14.162, -47.518, 112.71, 148.263, 50.786, -30.412, -175]
  MoveL 203 to (83, 1.72, -124.97) mm, rotated rx 42.04 ry 15.1 rz 65.25 deg; joints [-14.163, -47.52, 112.702, 148.258, 50.778, -30.405, -175]
  MoveL 204 to (83.07, 1.59, -125) mm, rotated rx 42.04 ry 15.1 rz 65.25 deg; joints [-14.163, -47.52, 112.692, 148.253, 50.769, -30.398, -175]
  MoveL 205 to (83.14, 1.29, -125.06) mm, rotated rx 42.04 ry 15.1 rz 65.25 deg; joints [-14.164, -47.515, 112.666, 148.244, 50.752, -30.384, -175]
  MoveL 206 to (83.1, 0.49, -125.19) mm, rotated rx 42.04 ry 15.1 rz 65.25 deg; joints [-14.163, -47.486, 112.597, 148.227, 50.717, -30.357, -175]
  MoveL 207 to (82.84, -0.48, -125.33) mm, rotated rx 42.04 ry 15.1 rz 65.25 deg; joints [-14.162, -47.438, 112.508, 148.211, 50.682, -30.329, -175]
  MoveL 208 to (81.94, -2.64, -125.6) mm, rotated rx 42.04 ry 15.1 rz 65.25 deg; joints [-14.158, -47.313, 112.307, 148.183, 50.617, -30.279, -175]
  MoveL 209 to (80.88, -4.81, -125.84) mm, rotated rx 42.04 ry 15.1 rz 65.25 deg; joints [-14.152, -47.178, 112.103, 148.16, 50.558, -30.235, -175]
  MoveL 210 to (56.65, -53.05, -130.92) mm, rotated rx 42.04 ry 15.1 rz 65.25 deg; joints [-14.023, -44.128, 107.47, 147.607, 49.186, -29.197, -175]
  MoveL 211 to (54.93, -56.48, -131.28) mm, rotated rx 42.04 ry 15.1 rz 65.25 deg; joints [-14.014, -43.91, 107.134, 147.563, 49.084, -29.117, -175]
  MoveL 212 to (53.09, -59.74, -131.7) mm, rotated rx 42.04 ry 15.1 rz 65.25 deg; joints [-14.008, -43.691, 106.808, 147.52, 48.993, -29.045, -175]
  MoveL 213 to (52.13, -60.88, -131.91) mm, rotated rx 42.04 ry 15.1 rz 65.25 deg; joints [-14.009, -43.595, 106.688, 147.508, 48.972, -29.027, -175]
  MoveL 214 to (51.68, -61.19, -132) mm, rotated rx 42.04 ry 15.1 rz 65.25 deg; joints [-14.01, -43.558, 106.651, 147.507, 48.974, -29.027, -175]
  MoveL 215 to (51.46, -61.26, -132.05) mm, rotated rx 42.04 ry 15.1 rz 65.25 deg; joints [-14.012, -43.542, 106.641, 147.508, 48.978, -29.03, -175]
  MoveL 216 to (51.25, -61.26, -132.09) mm, rotated rx 42.04 ry 15.1 rz 65.25 deg; joints [-14.013, -43.53, 106.636, 147.509, 48.985, -29.035, -175]
  MoveL 217 to (51.05, -61.2, -132.13) mm, rotated rx 42.04 ry 15.1 rz 65.25 deg; joints [-14.015, -43.52, 106.638, 147.513, 48.995, -29.042, -175]
  MoveL 218 to (50.86, -61.06, -132.16) mm, rotated rx 42.04 ry 15.1 rz 65.25 deg; joints [-14.017, -43.513, 106.646, 147.517, 49.008, -29.051, -175]
  MoveL 219 to (50.69, -60.85, -132.19) mm, rotated rx 42.04 ry 15.1 rz 65.25 deg; joints [-14.019, -43.51, 106.661, 147.523, 49.025, -29.063, -175]
  MoveL 220 to (50.52, -60.55, -132.22) mm, rotated rx 42.04 ry 15.1 rz 65.25 deg; joints [-14.022, -43.51, 106.684, 147.53, 49.045, -29.078, -175]
  MoveL 221 to (50.02, -58.41, -132.26) mm, rotated rx 42.04 ry 15.1 rz 65.25 deg; joints [-14.038, -43.551, 106.863, 147.575, 49.164, -29.168, -175]
  MoveL 222 to (49.77, -56.34, -132.26) mm, rotated rx 42.04 ry 15.1 rz 65.25 deg; joints [-14.051, -43.605, 107.041, 147.616, 49.273, -29.25, -175]
  MoveL 223 to (49.77, -52.53, -132.31) mm, rotated rx 42.04 ry 15.1 rz 65.25 deg; joints [-14.078, -43.729, 107.375, 147.68, 49.456, -29.384, -175]
  MoveL 224 to (50.54, -49.07, -132.42) mm, rotated rx 42.04 ry 15.1 rz 65.25 deg; joints [-14.105, -43.888, 107.69, 147.718, 49.594, -29.481, -175]
  MoveL 225 to (53.25, -43.66, -132.72) mm, rotated rx 42.04 ry 15.1 rz 65.25 deg; joints [-14.153, -44.223, 108.205, 147.741, 49.758, -29.583, -175]
  MoveL 226 to (54.73, -41.82, -132.85) mm, rotated rx 42.04 ry 15.1 rz 65.25 deg; joints [-14.171, -44.37, 108.389, 147.737, 49.793, -29.6, -175]
  MoveL 227 to (77.59, -15.62, -134.71) mm, rotated rx 42.04 ry 15.1 rz 65.25 deg; joints [-14.432, -46.577, 110.999, 147.602, 50.194, -29.756, -175]
  MoveL 228 to (79.53, -13.37, -134.87) mm, rotated rx 42.04 ry 15.1 rz 65.25 deg; joints [-14.454, -46.766, 111.219, 147.588, 50.226, -29.767, -175]
  MoveL 229 to (81.61, -10.27, -135.12) mm, rotated rx 42.04 ry 15.1 rz 65.25 deg; joints [-14.487, -46.99, 111.512, 147.58, 50.292, -29.8, -175]
  MoveL 230 to (82.14, -8.89, -135.26) mm, rotated rx 42.04 ry 15.1 rz 65.25 deg; joints [-14.502, -47.066, 111.636, 147.583, 50.336, -29.826, -175]
  MoveL 231 to (82.18, -8.34, -135.33) mm, rotated rx 42.04 ry 15.1 rz 65.25 deg; joints [-14.509, -47.085, 111.682, 147.587, 50.36, -29.842, -175]
  MoveL 232 to (82.13, -8.12, -135.36) mm, rotated rx 42.04 ry 15.1 rz 65.25 deg; joints [-14.512, -47.089, 111.699, 147.589, 50.372, -29.85, -175]
  MoveL 233 to (82.03, -7.94, -135.4) mm, rotated rx 42.04 ry 15.1 rz 65.25 deg; joints [-14.514, -47.088, 111.713, 147.592, 50.385, -29.858, -175]
  MoveL 234 to (81.87, -7.8, -135.43) mm, rotated rx 42.04 ry 15.1 rz 65.25 deg; joints [-14.517, -47.083, 111.722, 147.596, 50.397, -29.867, -175]
  MoveL 235 to (81.66, -7.7, -135.47) mm, rotated rx 42.04 ry 15.1 rz 65.25 deg; joints [-14.519, -47.073, 111.726, 147.6, 50.41, -29.876, -175]
  MoveL 236 to (81.38, -7.66, -135.5) mm, rotated rx 42.04 ry 15.1 rz 65.25 deg; joints [-14.52, -47.057, 111.725, 147.605, 50.422, -29.886, -175]
  MoveL 237 to (81.04, -7.67, -135.54) mm, rotated rx 42.04 ry 15.1 rz 65.25 deg; joints [-14.521, -47.036, 111.718, 147.61, 50.435, -29.895, -175]
  MoveL 238 to (78.95, -8.33, -135.66) mm, rotated rx 42.04 ry 15.1 rz 65.25 deg; joints [-14.521, -46.888, 111.628, 147.636, 50.484, -29.936, -175]
  MoveL 239 to (78.47, -8.53, -135.68) mm, rotated rx 42.04 ry 15.1 rz 65.25 deg; joints [-14.52, -46.852, 111.603, 147.642, 50.493, -29.944, -175]
  MoveL 240 to (78.06, -8.74, -135.73) mm, rotated rx 42.04 ry 15.1 rz 65.25 deg; joints [-14.52, -46.82, 111.578, 147.645, 50.499, -29.949, -175]
  MoveL 241 to (77.68, -8.96, -135.8) mm, rotated rx 42.04 ry 15.1 rz 65.25 deg; joints [-14.521, -46.79, 111.553, 147.645, 50.503, -29.951, -175]
  MoveL 242 to (77.28, -9.16, -135.86) mm, rotated rx 42.04 ry 15.1 rz 65.25 deg; joints [-14.522, -46.759, 111.528, 147.647, 50.509, -29.956, -175]
  MoveL 243 to (76.86, -9.36, -135.89) mm, rotated rx 42.04 ry 15.1 rz 65.25 deg; joints [-14.522, -46.727, 111.504, 147.651, 50.515, -29.961, -175]
  MoveL 244 to (72.52, -11.13, -135.9) mm, rotated rx 42.04 ry 15.1 rz 65.25 deg; joints [-14.508, -46.408, 111.285, 147.712, 50.597, -30.037, -175]
  MoveL 245 to (72.12, -11.31, -135.92) mm, rotated rx 42.04 ry 15.1 rz 65.25 deg; joints [-14.507, -46.377, 111.263, 147.716, 50.603, -30.043, -175]
  MoveL 246 to (71.68, -11.49, -135.93) mm, rotated rx 42.04 ry 15.1 rz 65.25 deg; joints [-14.506, -46.345, 111.24, 147.722, 50.611, -30.05, -175]
  MoveL 247 to (70.72, -11.88, -135.93) mm, rotated rx 42.04 ry 15.1 rz 65.25 deg; joints [-14.503, -46.274, 111.191, 147.735, 50.629, -30.066, -175]
  MoveL 248 to (70.2, -12.11, -135.94) mm, rotated rx 42.04 ry 15.1 rz 65.25 deg; joints [-14.502, -46.235, 111.163, 147.742, 50.638, -30.075, -175]
  MoveL 249 to (69.65, -12.36, -135.96) mm, rotated rx 42.04 ry 15.1 rz 65.25 deg; joints [-14.5, -46.194, 111.132, 147.748, 50.646, -30.082, -175]
  MoveL 250 to (69.07, -12.68, -135.99) mm, rotated rx 42.04 ry 15.1 rz 65.25 deg; joints [-14.499, -46.148, 111.095, 147.753, 50.653, -30.089, -175]
  MoveL 251 to (68.53, -13.06, -136.01) mm, rotated rx 42.04 ry 15.1 rz 65.25 deg; joints [-14.497, -46.103, 111.053, 147.757, 50.656, -30.092, -175]
  MoveL 252 to (68.02, -13.48, -136.03) mm, rotated rx 42.04 ry 15.1 rz 65.25 deg; joints [-14.494, -46.059, 111.009, 147.76, 50.655, -30.093, -175]
  MoveL 253 to (69.19, -12.88, -137.01) mm, rotated rx 42.04 ry 15.1 rz 65.25 deg; joints [-14.538, -46.143, 111.064, 147.695, 50.641, -30.053, -175]
  MoveL 254 to (68.73, -14.14, -137.43) mm, rotated rx 42.04 ry 15.1 rz 65.25 deg; joints [-14.546, -46.072, 110.943, 147.663, 50.6, -30.014, -175]
  MoveL 255 to (68.09, -15.49, -137.75) mm, rotated rx 42.04 ry 15.1 rz 65.25 deg; joints [-14.549, -45.989, 110.812, 147.639, 50.561, -29.981, -175]
  MoveL 256 to (67.25, -16.96, -137.99) mm, rotated rx 42.04 ry 15.1 rz 65.25 deg; joints [-14.548, -45.89, 110.669, 147.621, 50.523, -29.95, -175]
  MoveL 257 to (66.1, -18.76, -138.21) mm, rotated rx 42.04 ry 15.1 rz 65.25 deg; joints [-14.543, -45.761, 110.493, 147.605, 50.481, -29.919, -175]
  MoveL 258 to (64.92, -20.54, -138.32) mm, rotated rx 42.04 ry 15.1 rz 65.25 deg; joints [-14.535, -45.633, 110.319, 147.595, 50.441, -29.892, -175]
  MoveL 259 to (63.74, -22.32, -138.43) mm, rotated rx 42.04 ry 15.1 rz 65.25 deg; joints [-14.526, -45.504, 110.145, 147.585, 50.401, -29.864, -175]
  MoveL 260 to (62.57, -24.1, -138.66) mm, rotated rx 42.04 ry 15.1 rz 65.25 deg; joints [-14.522, -45.375, 109.968, 147.569, 50.36, -29.833, -175]
  MoveL 261 to (61.39, -25.88, -138.78) mm, rotated rx 42.04 ry 15.1 rz 65.25 deg; joints [-14.514, -45.247, 109.794, 147.558, 50.319, -29.805, -175]
  MoveL 262 to (60.21, -27.66, -139.01) mm, rotated rx 42.04 ry 15.1 rz 65.25 deg; joints [-14.51, -45.117, 109.617, 147.542, 50.278, -29.773, -175]
  MoveL 263 to (59.02, -29.43, -139.12) mm, rotated rx 42.04 ry 15.1 rz 65.25 deg; joints [-14.502, -44.988, 109.442, 147.531, 50.238, -29.745, -175]
  MoveL 264 to (57.83, -31.2, -139.24) mm, rotated rx 42.04 ry 15.1 rz 65.25 deg; joints [-14.494, -44.859, 109.267, 147.52, 50.197, -29.717, -175]
  MoveL 265 to (56.64, -32.97, -139.48) mm, rotated rx 42.04 ry 15.1 rz 65.25 deg; joints [-14.491, -44.729, 109.09, 147.503, 50.156, -29.686, -175]
  MoveL 266 to (55.48, -34.65, -139.58) mm, rotated rx 42.04 ry 15.1 rz 65.25 deg; joints [-14.483, -44.606, 108.923, 147.493, 50.118, -29.659, -175]
  MoveL 267 to (54.36, -36.29, -139.79) mm, rotated rx 42.04 ry 15.1 rz 65.25 deg; joints [-14.479, -44.484, 108.758, 147.478, 50.081, -29.63, -175]
  MoveL 268 to (53.04, -38.26, -139.95) mm, rotated rx 42.04 ry 15.1 rz 65.25 deg; joints [-14.471, -44.341, 108.562, 147.464, 50.034, -29.597, -175]
  MoveL 269 to (51.48, -40.49, -140.04) mm, rotated rx 42.04 ry 15.1 rz 65.25 deg; joints [-14.459, -44.175, 108.339, 147.453, 49.983, -29.563, -175]
  MoveL 270 to (50.32, -42.21, -140.1) mm, rotated rx 42.04 ry 15.1 rz 65.25 deg; joints [-14.449, -44.05, 108.168, 147.444, 49.942, -29.535, -175]
  MoveL 271 to (49.24, -43.8, -140.23) mm, rotated rx 42.04 ry 15.1 rz 65.25 deg; joints [-14.443, -43.933, 108.008, 147.432, 49.904, -29.508, -175]
  MoveL 272 to (48.12, -45.44, -140.34) mm, rotated rx 42.04 ry 15.1 rz 65.25 deg; joints [-14.435, -43.813, 107.844, 147.421, 49.866, -29.481, -175]
  MoveL 273 to (47.01, -47.05, -140.45) mm, rotated rx 42.04 ry 15.1 rz 65.25 deg; joints [-14.428, -43.694, 107.682, 147.41, 49.827, -29.453, -175]
  MoveL 274 to (45.85, -48.75, -140.52) mm, rotated rx 42.04 ry 15.1 rz 65.25 deg; joints [-14.419, -43.57, 107.511, 147.4, 49.787, -29.426, -175]
  MoveL 275 to (44.59, -50.58, -140.62) mm, rotated rx 42.04 ry 15.1 rz 65.25 deg; joints [-14.41, -43.435, 107.327, 147.389, 49.743, -29.395, -175]
  MoveL 276 to (43.19, -52.55, -140.88) mm, rotated rx 42.04 ry 15.1 rz 65.25 deg; joints [-14.406, -43.286, 107.125, 147.369, 49.697, -29.359, -175]
  MoveL 277 to (42.36, -54.62, -141.86) mm, rotated rx 42.04 ry 15.1 rz 65.25 deg; joints [-14.43, -43.163, 106.913, 147.299, 49.627, -29.284, -175]
  MoveL 278 to (42.38, -53.48, -142.35) mm, rotated rx 42.04 ry 15.1 rz 65.25 deg; joints [-14.457, -43.198, 107.005, 147.294, 49.682, -29.312, -175]
  MoveL 279 to (42.39, -52.89, -142.66) mm, rotated rx 42.04 ry 15.1 rz 65.25 deg; joints [-14.473, -43.216, 107.053, 147.288, 49.711, -29.326, -175]
  MoveL 280 to (42.38, -52.79, -142.81) mm, rotated rx 42.04 ry 15.1 rz 65.25 deg; joints [-14.479, -43.218, 107.059, 147.282, 49.716, -29.325, -175]
  MoveL 281 to (42.37, -53.13, -142.85) mm, rotated rx 42.04 ry 15.1 rz 65.25 deg; joints [-14.478, -43.206, 107.028, 147.274, 49.7, -29.312, -175]
  MoveL 282 to (42.37, -53.6, -142.86) mm, rotated rx 42.04 ry 15.1 rz 65.25 deg; joints [-14.476, -43.19, 106.987, 147.266, 49.678, -29.296, -175]
  MoveL 283 to (42.34, -54.08, -142.9) mm, rotated rx 42.04 ry 15.1 rz 65.25 deg; joints [-14.474, -43.173, 106.944, 147.256, 49.656, -29.278, -175]
  MoveL 284 to (42.31, -54.53, -142.96) mm, rotated rx 42.04 ry 15.1 rz 65.25 deg; joints [-14.473, -43.156, 106.903, 147.246, 49.635, -29.262, -175]
  MoveL 285 to (42.28, -54.99, -143) mm, rotated rx 42.04 ry 15.1 rz 65.25 deg; joints [-14.471, -43.139, 106.861, 147.237, 49.614, -29.245, -175]
  MoveL 286 to (42.26, -55.48, -143.02) mm, rotated rx 42.04 ry 15.1 rz 65.25 deg; joints [-14.469, -43.122, 106.818, 147.228, 49.591, -29.227, -175]
  MoveL 287 to (42.25, -58.1, -143.02) mm, rotated rx 42.04 ry 15.1 rz 65.25 deg; joints [-14.451, -43.036, 106.587, 147.182, 49.466, -29.133, -175]
  MoveL 288 to (42.24, -58.56, -143.04) mm, rotated rx 42.04 ry 15.1 rz 65.25 deg; joints [-14.449, -43.02, 106.546, 147.174, 49.445, -29.117, -175]
  MoveL 289 to (42.21, -58.94, -143.07) mm, rotated rx 42.04 ry 15.1 rz 65.25 deg; joints [-14.448, -43.005, 106.511, 147.166, 49.427, -29.103, -175]
  MoveL 290 to (42.19, -59.4, -143.09) mm, rotated rx 42.04 ry 15.1 rz 65.25 deg; joints [-14.445, -42.989, 106.47, 147.157, 49.405, -29.086, -175]
  MoveL 291 to (42.18, -60, -143.11) mm, rotated rx 42.04 ry 15.1 rz 65.25 deg; joints [-14.442, -42.968, 106.417, 147.146, 49.377, -29.064, -175]
  MoveL 292 to (42.13, -60.72, -143.17) mm, rotated rx 42.04 ry 15.1 rz 65.25 deg; joints [-14.439, -42.942, 106.352, 147.131, 49.344, -29.038, -175]
  MoveL 293 to (42.11, -61.34, -143.2) mm, rotated rx 42.04 ry 15.1 rz 65.25 deg; joints [-14.436, -42.92, 106.296, 147.119, 49.315, -29.016, -175]
  MoveL 294 to (42.11, -61.87, -143.2) mm, rotated rx 42.04 ry 15.1 rz 65.25 deg; joints [-14.433, -42.902, 106.249, 147.11, 49.29, -28.996, -175]
  MoveL 295 to (42.1, -63.44, -143.2) mm, rotated rx 42.04 ry 15.1 rz 65.25 deg; joints [-14.422, -42.849, 106.11, 147.082, 49.215, -28.939, -175]
  MoveL 296 to (41.79, -66.34, -143.54) mm, rotated rx 42.04 ry 15.1 rz 65.25 deg; joints [-14.416, -42.733, 105.843, 147.019, 49.086, -28.834, -175]
  MoveL 297 to (41.42, -67.58, -143.97) mm, rotated rx 42.04 ry 15.1 rz 65.25 deg; joints [-14.424, -42.667, 105.719, 146.982, 49.04, -28.788, -175]
  MoveL 298 to (40.9, -68.68, -144.57) mm, rotated rx 42.04 ry 15.1 rz 65.25 deg; joints [-14.439, -42.596, 105.603, 146.941, 49.006, -28.748, -175]
  MoveL 299 to (39.42, -70.47, -146.28) mm, rotated rx 42.04 ry 15.1 rz 65.25 deg; joints [-14.492, -42.439, 105.39, 146.851, 48.972, -28.681, -175]
  MoveL 300 to (37.35, -71.7, -148.68) mm, rotated rx 42.04 ry 15.1 rz 65.25 deg; joints [-14.574, -42.261, 105.204, 146.746, 48.986, -28.633, -175]
  MoveL 301 to (35.34, -72.15, -151.07) mm, rotated rx 42.04 ry 15.1 rz 65.25 deg; joints [-14.661, -42.113, 105.088, 146.655, 49.035, -28.613, -175]
  MoveL 302 to (34.6, -71.99, -152.01) mm, rotated rx 42.04 ry 15.1 rz 65.25 deg; joints [-14.698, -42.068, 105.073, 146.625, 49.069, -28.617, -175]
  MoveL 303 to (34.02, -71.57, -152.78) mm, rotated rx 42.04 ry 15.1 rz 65.25 deg; joints [-14.73, -42.044, 105.087, 146.604, 49.109, -28.629, -175]
  MoveL 304 to (33.8, -71.26, -153.1) mm, rotated rx 42.04 ry 15.1 rz 65.25 deg; joints [-14.744, -42.039, 105.105, 146.598, 49.132, -28.638, -175]
  MoveL 305 to (33.63, -70.89, -153.38) mm, rotated rx 42.04 ry 15.1 rz 65.25 deg; joints [-14.757, -42.039, 105.13, 146.594, 49.156, -28.65, -175]
  MoveL 306 to (33.4, -69.96, -153.81) mm, rotated rx 42.04 ry 15.1 rz 65.25 deg; joints [-14.78, -42.054, 105.202, 146.593, 49.209, -28.68, -175]
  MoveL 307 to (33.35, -68.77, -154.07) mm, rotated rx 42.04 ry 15.1 rz 65.25 deg; joints [-14.798, -42.088, 105.302, 146.603, 49.268, -28.719, -175]
  MoveL 308 to (33.47, -67.32, -154.15) mm, rotated rx 42.04 ry 15.1 rz 65.25 deg; joints [-14.811, -42.143, 105.431, 146.622, 49.334, -28.767, -175]
  MoveL 309 to (33.54, -66.8, -154.15) mm, rotated rx 42.04 ry 15.1 rz 65.25 deg; joints [-14.815, -42.164, 105.479, 146.63, 49.357, -28.784, -175]
  MoveL 310 to (33.64, -66.37, -154.1) mm, rotated rx 42.04 ry 15.1 rz 65.25 deg; joints [-14.816, -42.184, 105.519, 146.639, 49.374, -28.798, -175]
  MoveL 311 to (33.74, -65.95, -154.04) mm, rotated rx 42.04 ry 15.1 rz 65.25 deg; joints [-14.816, -42.204, 105.56, 146.647, 49.391, -28.813, -175]
  MoveL 312 to (33.82, -65.49, -154) mm, rotated rx 42.04 ry 15.1 rz 65.25 deg; joints [-14.818, -42.225, 105.603, 146.656, 49.41, -28.828, -175]
  MoveL 313 to (33.9, -65, -153.98) mm, rotated rx 42.04 ry 15.1 rz 65.25 deg; joints [-14.821, -42.246, 105.648, 146.664, 49.431, -28.844, -175]
  MoveL 314 to (33.98, -64.47, -153.98) mm, rotated rx 42.04 ry 15.1 rz 65.25 deg; joints [-14.824, -42.267, 105.697, 146.672, 49.454, -28.862, -175]
  MoveL 315 to (34.05, -63.95, -153.98) mm, rotated rx 42.04 ry 15.1 rz 65.25 deg; joints [-14.828, -42.288, 105.744, 146.68, 49.477, -28.879, -175]
  MoveL 316 to (34.1, -63.44, -153.99) mm, rotated rx 42.04 ry 15.1 rz 65.25 deg; joints [-14.832, -42.308, 105.789, 146.687, 49.5, -28.895, -175]
  MoveL 317 to (34.16, -62.95, -154) mm, rotated rx 42.04 ry 15.1 rz 65.25 deg; joints [-14.836, -42.327, 105.834, 146.694, 49.522, -28.912, -175]
  MoveL 318 to (34.23, -62.49, -153.98) mm, rotated rx 42.04 ry 15.1 rz 65.25 deg; joints [-14.838, -42.347, 105.876, 146.702, 49.541, -28.927, -175]
  MoveL 319 to (34.31, -62.04, -153.94) mm, rotated rx 42.04 ry 15.1 rz 65.25 deg; joints [-14.84, -42.367, 105.918, 146.71, 49.56, -28.942, -175]
  MoveL 320 to (34.42, -61.5, -153.89) mm, rotated rx 42.04 ry 15.1 rz 65.25 deg; joints [-14.842, -42.391, 105.968, 146.72, 49.582, -28.96, -175]
  MoveL 321 to (34.55, -60.81, -153.84) mm, rotated rx 42.04 ry 15.1 rz 65.25 deg; joints [-14.845, -42.422, 106.033, 146.732, 49.611, -28.983, -175]
  MoveL 322 to (34.66, -60.18, -153.81) mm, rotated rx 42.04 ry 15.1 rz 65.25 deg; joints [-14.848, -42.449, 106.091, 146.743, 49.638, -29.003, -175]
  MoveL 323 to (35.01, -57.58, -153.81) mm, rotated rx 42.04 ry 15.1 rz 65.25 deg; joints [-14.867, -42.554, 106.326, 146.781, 49.751, -29.088, -175]
  MoveL 324 to (35.11, -56.96, -153.78) mm, rotated rx 42.04 ry 15.1 rz 65.25 deg; joints [-14.869, -42.58, 106.383, 146.792, 49.777, -29.109, -175]
  MoveL 325 to (35.21, -56.41, -153.72) mm, rotated rx 42.04 ry 15.1 rz 65.25 deg; joints [-14.871, -42.604, 106.434, 146.802, 49.801, -29.127, -175]
  MoveL 326 to (35.25, -56.21, -153.57) mm, rotated rx 42.04 ry 15.1 rz 65.25 deg; joints [-14.867, -42.615, 106.455, 146.812, 49.809, -29.137, -175]
  MoveL 327 to (35.23, -56.33, -153.31) mm, rotated rx 42.04 ry 15.1 rz 65.25 deg; joints [-14.856, -42.611, 106.448, 146.824, 49.803, -29.14, -175]
  MoveL 328 to (35.13, -56.78, -152.9) mm, rotated rx 42.04 ry 15.1 rz 65.25 deg; joints [-14.837, -42.594, 106.414, 146.839, 49.784, -29.137, -175]
  MoveL 329 to (36.15, -56.59, -152.1) mm, rotated rx 42.04 ry 15.1 rz 65.25 deg; joints [-14.808, -42.665, 106.463, 146.863, 49.759, -29.135, -175]
  MoveL 330 to (37.5, -55.14, -151.88) mm, rotated rx 42.04 ry 15.1 rz 65.25 deg; joints [-14.81, -42.794, 106.619, 146.873, 49.782, -29.153, -175]
  MoveL 331 to (38.85, -53.66, -151.72) mm, rotated rx 42.04 ry 15.1 rz 65.25 deg; joints [-14.815, -42.923, 106.776, 146.881, 49.807, -29.171, -175]
  MoveL 332 to (40.23, -52.13, -151.57) mm, rotated rx 42.04 ry 15.1 rz 65.25 deg; joints [-14.821, -43.055, 106.938, 146.888, 49.833, -29.19, -175]
  MoveL 333 to (41.5, -50.75, -151.28) mm, rotated rx 42.04 ry 15.1 rz 65.25 deg; joints [-14.82, -43.177, 107.087, 146.902, 49.856, -29.21, -175]
  MoveL 334 to (42.91, -49.19, -151.09) mm, rotated rx 42.04 ry 15.1 rz 65.25 deg; joints [-14.824, -43.313, 107.253, 146.91, 49.882, -29.229, -175]
  MoveL 335 to (44.4, -47.54, -150.9) mm, rotated rx 42.04 ry 15.1 rz 65.25 deg; joints [-14.829, -43.456, 107.427, 146.918, 49.909, -29.249, -175]
  MoveL 336 to (45.9, -45.87, -150.82) mm, rotated rx 42.04 ry 15.1 rz 65.25 deg; joints [-14.838, -43.599, 107.601, 146.922, 49.937, -29.266, -175]
  MoveL 337 to (47.71, -43.83, -150.73) mm, rotated rx 42.04 ry 15.1 rz 65.25 deg; joints [-14.85, -43.774, 107.813, 146.925, 49.971, -29.288, -175]
  MoveL 338 to (49.01, -42.36, -150.62) mm, rotated rx 42.04 ry 15.1 rz 65.25 deg; joints [-14.857, -43.899, 107.966, 146.929, 49.996, -29.304, -175]
  MoveL 339 to (50.22, -41, -150.41) mm, rotated rx 42.04 ry 15.1 rz 65.25 deg; joints [-14.859, -44.017, 108.11, 146.939, 50.018, -29.322, -175]
  MoveL 340 to (51.55, -39.48, -150.22) mm, rotated rx 42.04 ry 15.1 rz 65.25 deg; joints [-14.862, -44.146, 108.268, 146.947, 50.043, -29.34, -175]
  MoveL 341 to (52.96, -37.88, -150.1) mm, rotated rx 42.04 ry 15.1 rz 65.25 deg; joints [-14.87, -44.283, 108.434, 146.951, 50.069, -29.357, -175]
  MoveL 342 to (54.35, -36.29, -149.92) mm, rotated rx 42.04 ry 15.1 rz 65.25 deg; joints [-14.875, -44.419, 108.599, 146.959, 50.095, -29.376, -175]
  MoveL 343 to (55.74, -34.7, -149.8) mm, rotated rx 42.04 ry 15.1 rz 65.25 deg; joints [-14.882, -44.554, 108.763, 146.963, 50.121, -29.393, -175]
  MoveL 344 to (57.17, -33.05, -149.62) mm, rotated rx 42.04 ry 15.1 rz 65.25 deg; joints [-14.887, -44.693, 108.933, 146.97, 50.148, -29.412, -175]
  MoveL 345 to (58.57, -31.44, -149.5) mm, rotated rx 42.04 ry 15.1 rz 65.25 deg; joints [-14.895, -44.83, 109.098, 146.974, 50.174, -29.429, -175]
  MoveL 346 to (59.96, -29.82, -149.27) mm, rotated rx 42.04 ry 15.1 rz 65.25 deg; joints [-14.898, -44.966, 109.265, 146.985, 50.2, -29.449, -175]
  MoveL 347 to (61.36, -28.2, -149.16) mm, rotated rx 42.04 ry 15.1 rz 65.25 deg; joints [-14.906, -45.103, 109.43, 146.988, 50.226, -29.465, -175]
  MoveL 348 to (62.75, -26.59, -149.04) mm, rotated rx 42.04 ry 15.1 rz 65.25 deg; joints [-14.914, -45.239, 109.595, 146.992, 50.251, -29.482, -175]
  MoveL 349 to (64.13, -24.95, -148.82) mm, rotated rx 42.04 ry 15.1 rz 65.25 deg; joints [-14.917, -45.376, 109.762, 147.001, 50.278, -29.502, -175]
  MoveL 350 to (65.34, -23.44, -148.61) mm, rotated rx 42.04 ry 15.1 rz 65.25 deg; joints [-14.921, -45.498, 109.915, 147.011, 50.305, -29.522, -175]
  MoveL 351 to (66.39, -22.03, -148.32) mm, rotated rx 42.04 ry 15.1 rz 65.25 deg; joints [-14.92, -45.609, 110.059, 147.027, 50.332, -29.546, -175]
  MoveL 352 to (67.29, -20.67, -147.92) mm, rotated rx 42.04 ry 15.1 rz 65.25 deg; joints [-14.914, -45.71, 110.197, 147.05, 50.362, -29.575, -175]
  MoveL 353 to (65.98, -21.37, -146.99) mm, rotated rx 42.04 ry 15.1 rz 65.25 deg; joints [-14.872, -45.614, 110.13, 147.114, 50.376, -29.614, -175]
  MoveL 354 to (66.44, -21.02, -146.98) mm, rotated rx 42.04 ry 15.1 rz 65.25 deg; joints [-14.874, -45.653, 110.167, 147.11, 50.375, -29.612, -175]
  MoveL 355 to (66.89, -20.74, -146.96) mm, rotated rx 42.04 ry 15.1 rz 65.25 deg; joints [-14.876, -45.69, 110.2, 147.107, 50.372, -29.609, -175]
  MoveL 356 to (67.31, -20.52, -146.9) mm, rotated rx 42.04 ry 15.1 rz 65.25 deg; joints [-14.875, -45.722, 110.226, 147.105, 50.367, -29.605, -175]
  MoveL 357 to (67.71, -20.33, -146.83) mm, rotated rx 42.04 ry 15.1 rz 65.25 deg; joints [-14.874, -45.753, 110.25, 147.103, 50.361, -29.601, -175]
  MoveL 358 to (68.15, -20.17, -146.78) mm, rotated rx 42.04 ry 15.1 rz 65.25 deg; joints [-14.873, -45.785, 110.272, 147.099, 50.352, -29.594, -175]
  MoveL 359 to (68.61, -20.02, -146.75) mm, rotated rx 42.04 ry 15.1 rz 65.25 deg; joints [-14.873, -45.818, 110.293, 147.094, 50.342, -29.585, -175]
  MoveL 360 to (69.12, -19.87, -146.73) mm, rotated rx 42.04 ry 15.1 rz 65.25 deg; joints [-14.874, -45.853, 110.314, 147.087, 50.33, -29.575, -175]
  MoveL 361 to (69.63, -19.74, -146.73) mm, rotated rx 42.04 ry 15.1 rz 65.25 deg; joints [-14.875, -45.887, 110.333, 147.079, 50.318, -29.564, -175]
  MoveL 362 to (70.08, -19.61, -146.72) mm, rotated rx 42.04 ry 15.1 rz 65.25 deg; joints [-14.876, -45.919, 110.352, 147.072, 50.308, -29.554, -175]
  MoveL 363 to (70.48, -19.48, -146.69) mm, rotated rx 42.04 ry 15.1 rz 65.25 deg; joints [-14.876, -45.947, 110.37, 147.067, 50.299, -29.547, -175]
  MoveL 364 to (70.94, -19.34, -146.68) mm, rotated rx 42.04 ry 15.1 rz 65.25 deg; joints [-14.877, -45.98, 110.389, 147.06, 50.288, -29.537, -175]
  MoveL 365 to (71.45, -19.21, -146.68) mm, rotated rx 42.04 ry 15.1 rz 65.25 deg; joints [-14.878, -46.014, 110.409, 147.052, 50.276, -29.526, -175]
  MoveL 366 to (72.04, -19.04, -146.66) mm, rotated rx 42.04 ry 15.1 rz 65.25 deg; joints [-14.879, -46.055, 110.433, 147.044, 50.262, -29.514, -175]
  MoveL 367 to (72.7, -18.85, -146.62) mm, rotated rx 42.04 ry 15.1 rz 65.25 deg; joints [-14.879, -46.102, 110.461, 147.035, 50.246, -29.501, -175]
  MoveL 368 to (73.29, -18.68, -146.6) mm, rotated rx 42.04 ry 15.1 rz 65.25 deg; joints [-14.879, -46.143, 110.485, 147.027, 50.232, -29.489, -175]
  MoveL 369 to (73.9, -18.5, -146.57) mm, rotated rx 42.04 ry 15.1 rz 65.25 deg; joints [-14.88, -46.186, 110.511, 147.018, 50.218, -29.476, -175]
  MoveL 370 to (74.58, -18.29, -146.53) mm, rotated rx 42.04 ry 15.1 rz 65.25 deg; joints [-14.88, -46.234, 110.541, 147.01, 50.203, -29.463, -175]
  MoveL 371 to (75.15, -18.12, -146.52) mm, rotated rx 42.04 ry 15.1 rz 65.25 deg; joints [-14.881, -46.273, 110.564, 147.001, 50.189, -29.451, -175]
  MoveL 372 to (75.68, -17.98, -146.52) mm, rotated rx 42.04 ry 15.1 rz 65.25 deg; joints [-14.882, -46.309, 110.584, 146.993, 50.176, -29.439, -175]
  MoveL 373 to (77.2, -17.58, -146.52) mm, rotated rx 42.04 ry 15.1 rz 65.25 deg; joints [-14.886, -46.414, 110.642, 146.967, 50.138, -29.405, -175]
  MoveL 374 to (78.62, -17.28, -146.6) mm, rotated rx 42.04 ry 15.1 rz 65.25 deg; joints [-14.892, -46.508, 110.689, 146.938, 50.1, -29.368, -175]
  MoveL 375 to (79.8, -17.18, -146.85) mm, rotated rx 42.04 ry 15.1 rz 65.25 deg; joints [-14.903, -46.581, 110.711, 146.902, 50.06, -29.327, -175]
  MoveL 376 to (80.75, -17.29, -147.28) mm, rotated rx 42.04 ry 15.1 rz 65.25 deg; joints [-14.92, -46.632, 110.71, 146.858, 50.021, -29.282, -175]
  MoveL 377 to (81.14, -17.42, -147.55) mm, rotated rx 42.04 ry 15.1 rz 65.25 deg; joints [-14.93, -46.649, 110.701, 146.834, 50.001, -29.258, -175]
  MoveL 378 to (81.47, -17.6, -147.87) mm, rotated rx 42.04 ry 15.1 rz 65.25 deg; joints [-14.941, -46.661, 110.685, 146.807, 49.981, -29.233, -175]
  MoveL 379 to (81.96, -18.11, -148.63) mm, rotated rx 42.04 ry 15.1 rz 65.25 deg; joints [-14.968, -46.668, 110.637, 146.75, 49.94, -29.18, -175]
  MoveL 380 to (82.21, -18.83, -149.55) mm, rotated rx 42.04 ry 15.1 rz 65.25 deg; joints [-14.999, -46.653, 110.564, 146.685, 49.9, -29.124, -175]
  MoveL 381 to (82.01, -20.88, -151.92) mm, rotated rx 42.04 ry 15.1 rz 65.25 deg; joints [-15.078, -46.558, 110.347, 146.534, 49.817, -28.998, -175]
  MoveL 382 to (81.03, -23.07, -154.28) mm, rotated rx 42.04 ry 15.1 rz 65.25 deg; joints [-15.154, -46.412, 110.105, 146.397, 49.756, -28.892, -175]
  MoveL 383 to (79.44, -24.76, -155.97) mm, rotated rx 42.04 ry 15.1 rz 65.25 deg; joints [-15.207, -46.249, 109.908, 146.316, 49.74, -28.841, -175]
  MoveL 384 to (78.41, -25.41, -156.56) mm, rotated rx 42.04 ry 15.1 rz 65.25 deg; joints [-15.225, -46.162, 109.826, 146.297, 49.749, -28.836, -175]
  MoveL 385 to (77.22, -25.94, -156.98) mm, rotated rx 42.04 ry 15.1 rz 65.25 deg; joints [-15.237, -46.071, 109.756, 146.292, 49.769, -28.845, -175]
  MoveL 386 to (74.38, -26.6, -157.32) mm, rotated rx 42.04 ry 15.1 rz 65.25 deg; joints [-15.244, -45.878, 109.649, 146.324, 49.842, -28.905, -175]
  MoveL 387 to (70.23, -27.14, -157.32) mm, rotated rx 42.04 ry 15.1 rz 65.25 deg; joints [-15.238, -45.613, 109.536, 146.402, 49.968, -29.018, -175]
  MoveL 388 to (69.68, -27.22, -157.34) mm, rotated rx 42.04 ry 15.1 rz 65.25 deg; joints [-15.238, -45.577, 109.52, 146.411, 49.983, -29.032, -175]
  MoveL 389 to (69.16, -27.32, -157.37) mm, rotated rx 42.04 ry 15.1 rz 65.25 deg; joints [-15.239, -45.543, 109.502, 146.418, 49.998, -29.044, -175]
  MoveL 390 to (68.64, -27.43, -157.44) mm, rotated rx 42.04 ry 15.1 rz 65.25 deg; joints [-15.24, -45.508, 109.483, 146.424, 50.011, -29.055, -175]
  MoveL 391 to (68.14, -27.55, -157.52) mm, rotated rx 42.04 ry 15.1 rz 65.25 deg; joints [-15.242, -45.473, 109.463, 146.428, 50.024, -29.064, -175]
  MoveL 392 to (67.65, -27.67, -157.6) mm, rotated rx 42.04 ry 15.1 rz 65.25 deg; joints [-15.244, -45.439, 109.443, 146.433, 50.036, -29.074, -175]
  MoveL 393 to (67.17, -27.76, -157.64) mm, rotated rx 42.04 ry 15.1 rz 65.25 deg; joints [-15.245, -45.408, 109.427, 146.439, 50.049, -29.084, -175]
  MoveL 394 to (66.7, -27.83, -157.65) mm, rotated rx 42.04 ry 15.1 rz 65.25 deg; joints [-15.245, -45.377, 109.413, 146.447, 50.063, -29.096, -175]
  MoveL 395 to (66.18, -27.9, -157.65) mm, rotated rx 42.04 ry 15.1 rz 65.25 deg; joints [-15.244, -45.344, 109.399, 146.457, 50.079, -29.11, -175]
  MoveL 396 to (65.56, -28, -157.69) mm, rotated rx 42.04 ry 15.1 rz 65.25 deg; joints [-15.244, -45.303, 109.379, 146.466, 50.096, -29.125, -175]
  MoveL 397 to (64.89, -28.13, -157.75) mm, rotated rx 42.04 ry 15.1 rz 65.25 deg; joints [-15.245, -45.259, 109.356, 146.475, 50.115, -29.141, -175]
  MoveL 398 to (64.3, -28.24, -157.77) mm, rotated rx 42.04 ry 15.1 rz 65.25 deg; joints [-15.245, -45.22, 109.336, 146.484, 50.13, -29.154, -175]
  MoveL 399 to (63.77, -28.39, -157.78) mm, rotated rx 42.04 ry 15.1 rz 65.25 deg; joints [-15.244, -45.183, 109.315, 146.492, 50.143, -29.166, -175]
  MoveL 400 to (63.25, -28.58, -157.78) mm, rotated rx 42.04 ry 15.1 rz 65.25 deg; joints [-15.242, -45.146, 109.289, 146.499, 50.152, -29.175, -175]
  MoveL 401 to (62.76, -28.89, -157.78) mm, rotated rx 42.04 ry 15.1 rz 65.25 deg; joints [-15.24, -45.107, 109.255, 146.504, 50.155, -29.179, -175]
  MoveL 402 to (62.28, -29.27, -157.78) mm, rotated rx 42.04 ry 15.1 rz 65.25 deg; joints [-15.237, -45.066, 109.214, 146.508, 50.154, -29.181, -175]
  MoveL 403 to (63.7, -28.59, -158.74) mm, rotated rx 42.04 ry 15.1 rz 65.25 deg; joints [-15.28, -45.166, 109.281, 146.441, 50.137, -29.136, -175]
  MoveL 404 to (62.93, -29.57, -159.16) mm, rotated rx 42.04 ry 15.1 rz 65.25 deg; joints [-15.289, -45.086, 109.176, 146.419, 50.119, -29.115, -175]
  MoveL 405 to (61.98, -30.62, -159.49) mm, rotated rx 42.04 ry 15.1 rz 65.25 deg; joints [-15.293, -44.993, 109.064, 146.405, 50.105, -29.099, -175]
  MoveL 406 to (60.84, -31.75, -159.74) mm, rotated rx 42.04 ry 15.1 rz 65.25 deg; joints [-15.294, -44.886, 108.943, 146.397, 50.093, -29.088, -175]
  MoveL 407 to (59.25, -33.17, -159.85) mm, rotated rx 42.04 ry 15.1 rz 65.25 deg; joints [-15.287, -44.745, 108.791, 146.401, 50.082, -29.084, -175]
  MoveL 408 to (57.68, -34.61, -160.08) mm, rotated rx 42.04 ry 15.1 rz 65.25 deg; joints [-15.285, -44.603, 108.636, 146.398, 50.071, -29.076, -175]
  MoveL 409 to (56.09, -36.03, -160.19) mm, rotated rx 42.04 ry 15.1 rz 65.25 deg; joints [-15.278, -44.461, 108.484, 146.401, 50.06, -29.071, -175]
  MoveL 410 to (54.49, -37.45, -160.31) mm, rotated rx 42.04 ry 15.1 rz 65.25 deg; joints [-15.271, -44.319, 108.331, 146.404, 50.05, -29.066, -175]
  MoveL 411 to (52.91, -38.87, -160.54) mm, rotated rx 42.04 ry 15.1 rz 65.25 deg; joints [-15.269, -44.177, 108.176, 146.4, 50.038, -29.058, -175]
  MoveL 412 to (51.31, -40.28, -160.66) mm, rotated rx 42.04 ry 15.1 rz 65.25 deg; joints [-15.262, -44.036, 108.023, 146.403, 50.027, -29.053, -175]
  MoveL 413 to (49.71, -41.7, -160.78) mm, rotated rx 42.04 ry 15.1 rz 65.25 deg; joints [-15.256, -43.894, 107.87, 146.405, 50.016, -29.048, -175]
  MoveL 414 to (47.87, -43.33, -160.94) mm, rotated rx 42.04 ry 15.1 rz 65.25 deg; joints [-15.249, -43.731, 107.693, 146.407, 50.003, -29.041, -175]
  MoveL 415 to (46.29, -44.71, -161.14) mm, rotated rx 42.04 ry 15.1 rz 65.25 deg; joints [-15.246, -43.591, 107.541, 146.405, 49.992, -29.034, -175]
  MoveL 416 to (44.55, -46.23, -161.33) mm, rotated rx 42.04 ry 15.1 rz 65.25 deg; joints [-15.242, -43.437, 107.373, 146.404, 49.979, -29.026, -175]
  MoveL 417 to (42.84, -47.72, -161.59) mm, rotated rx 42.04 ry 15.1 rz 65.25 deg; joints [-15.24, -43.286, 107.208, 146.4, 49.967, -29.017, -175]
  MoveL 418 to (41.24, -49.12, -161.71) mm, rotated rx 42.04 ry 15.1 rz 65.25 deg; joints [-15.233, -43.144, 107.054, 146.402, 49.955, -29.011, -175]
  MoveL 419 to (39.63, -50.52, -161.71) mm, rotated rx 42.04 ry 15.1 rz 65.25 deg; joints [-15.222, -43.004, 106.902, 146.409, 49.943, -29.007, -175]
  MoveL 420 to (38.04, -51.9, -161.78) mm, rotated rx 42.04 ry 15.1 rz 65.25 deg; joints [-15.215, -42.864, 106.75, 146.413, 49.931, -29.002, -175]
  MoveL 421 to (36.47, -53.24, -162) mm, rotated rx 42.04 ry 15.1 rz 65.25 deg; joints [-15.212, -42.727, 106.6, 146.41, 49.92, -28.995, -175]
  MoveL 422 to (34.71, -54.71, -162.35) mm, rotated rx 42.04 ry 15.1 rz 65.25 deg; joints [-15.214, -42.572, 106.431, 146.401, 49.909, -28.984, -175]
  MoveL 423 to (33.32, -55.87, -162.56) mm, rotated rx 42.04 ry 15.1 rz 65.25 deg; joints [-15.213, -42.451, 106.3, 146.398, 49.9, -28.976, -175]
  MoveL 424 to (31.42, -57.43, -162.86) mm, rotated rx 42.04 ry 15.1 rz 65.25 deg; joints [-15.213, -42.286, 106.122, 146.392, 49.889, -28.967, -175]
  MoveL 425 to (29.74, -58.86, -162.96) mm, rotated rx 42.04 ry 15.1 rz 65.25 deg; joints [-15.205, -42.139, 105.962, 146.395, 49.876, -28.961, -175]
  MoveL 426 to (28.14, -60.26, -162.98) mm, rotated rx 42.04 ry 15.1 rz 65.25 deg; joints [-15.195, -41.999, 105.807, 146.4, 49.861, -28.955, -175]
  MoveL 427 to (27.25, -60.37, -163.77) mm, rotated rx 42.04 ry 15.1 rz 65.25 deg; joints [-15.224, -41.938, 105.767, 146.375, 49.886, -28.957, -175]
  MoveL 428 to (27.44, -59.97, -164.16) mm, rotated rx 42.04 ry 15.1 rz 65.25 deg; joints [-15.242, -41.959, 105.799, 146.359, 49.899, -28.956, -175]
  MoveL 429 to (27.51, -59.85, -164.4) mm, rotated rx 42.04 ry 15.1 rz 65.25 deg; joints [-15.252, -41.966, 105.807, 146.347, 49.903, -28.952, -175]
  MoveL 430 to (27.47, -59.99, -164.53) mm, rotated rx 42.04 ry 15.1 rz 65.25 deg; joints [-15.256, -41.958, 105.792, 146.339, 49.898, -28.945, -175]
  MoveL 431 to (27.36, -60.37, -164.55) mm, rotated rx 42.04 ry 15.1 rz 65.25 deg; joints [-15.254, -41.939, 105.756, 146.334, 49.883, -28.934, -175]
  MoveL 432 to (27.23, -60.82, -164.56) mm, rotated rx 42.04 ry 15.1 rz 65.25 deg; joints [-15.251, -41.917, 105.714, 146.328, 49.866, -28.921, -175]
  MoveL 433 to (26.82, -62.33, -164.56) mm, rotated rx 42.04 ry 15.1 rz 65.25 deg; joints [-15.24, -41.843, 105.572, 146.309, 49.806, -28.876, -175]
  MoveL 434 to (26.67, -62.87, -164.58) mm, rotated rx 42.04 ry 15.1 rz 65.25 deg; joints [-15.237, -41.817, 105.522, 146.302, 49.786, -28.861, -175]
  MoveL 435 to (26.49, -63.39, -164.62) mm, rotated rx 42.04 ry 15.1 rz 65.25 deg; joints [-15.235, -41.789, 105.471, 146.294, 49.766, -28.845, -175]
  MoveL 436 to (26.29, -63.93, -164.7) mm, rotated rx 42.04 ry 15.1 rz 65.25 deg; joints [-15.234, -41.76, 105.419, 146.284, 49.747, -28.829, -175]
  MoveL 437 to (26.11, -64.45, -164.76) mm, rotated rx 42.04 ry 15.1 rz 65.25 deg; joints [-15.232, -41.731, 105.368, 146.275, 49.727, -28.813, -175]
  MoveL 438 to (25.96, -64.96, -164.79) mm, rotated rx 42.04 ry 15.1 rz 65.25 deg; joints [-15.23, -41.706, 105.319, 146.268, 49.708, -28.798, -175]
  MoveL 439 to (25.82, -65.43, -164.81) mm, rotated rx 42.04 ry 15.1 rz 65.25 deg; joints [-15.227, -41.682, 105.274, 146.261, 49.69, -28.784, -175]
  MoveL 440 to (25.67, -65.87, -164.85) mm, rotated rx 42.04 ry 15.1 rz 65.25 deg; joints [-15.225, -41.658, 105.232, 146.254, 49.674, -28.771, -175]
  MoveL 441 to (25.53, -66.29, -164.89) mm, rotated rx 42.04 ry 15.1 rz 65.25 deg; joints [-15.224, -41.636, 105.192, 146.247, 49.658, -28.758, -175]
  MoveL 442 to (25.39, -66.76, -164.91) mm, rotated rx 42.04 ry 15.1 rz 65.25 deg; joints [-15.221, -41.612, 105.146, 146.241, 49.639, -28.744, -175]
  MoveL 443 to (25.22, -67.33, -164.93) mm, rotated rx 42.04 ry 15.1 rz 65.25 deg; joints [-15.217, -41.584, 105.093, 146.233, 49.618, -28.727, -175]
  MoveL 444 to (25, -67.99, -164.98) mm, rotated rx 42.04 ry 15.1 rz 65.25 deg; joints [-15.215, -41.549, 105.029, 146.223, 49.593, -28.707, -175]
  MoveL 445 to (24.82, -68.57, -165.01) mm, rotated rx 42.04 ry 15.1 rz 65.25 deg; joints [-15.211, -41.519, 104.973, 146.214, 49.571, -28.69, -175]
  MoveL 446 to (24.28, -70.6, -165.01) mm, rotated rx 42.04 ry 15.1 rz 65.25 deg; joints [-15.197, -41.421, 104.782, 146.188, 49.49, -28.63, -175]
  MoveL 447 to (23.25, -73.33, -165.34) mm, rotated rx 42.04 ry 15.1 rz 65.25 deg; joints [-15.189, -41.269, 104.514, 146.142, 49.392, -28.548, -175]
  MoveL 448 to (22.58, -74.43, -165.75) mm, rotated rx 42.04 ry 15.1 rz 65.25 deg; joints [-15.197, -41.19, 104.395, 146.114, 49.36, -28.515, -175]
  MoveL 449 to (21.81, -75.37, -166.33) mm, rotated rx 42.04 ry 15.1 rz 65.25 deg; joints [-15.211, -41.11, 104.286, 146.082, 49.34, -28.487, -175]
  MoveL 450 to (19.95, -76.73, -167.98) mm, rotated rx 42.04 ry 15.1 rz 65.25 deg; joints [-15.263, -40.944, 104.1, 146.009, 49.336, -28.446, -175]
  MoveL 451 to (17.67, -77.41, -170.29) mm, rotated rx 42.04 ry 15.1 rz 65.25 deg; joints [-15.344, -40.772, 103.954, 145.923, 49.378, -28.425, -175]
  MoveL 452 to (15.64, -77.34, -172.59) mm, rotated rx 42.04 ry 15.1 rz 65.25 deg; joints [-15.431, -40.64, 103.879, 145.846, 49.447, -28.425, -175]
  MoveL 453 to (14.98, -76.99, -173.5) mm, rotated rx 42.04 ry 15.1 rz 65.25 deg; joints [-15.467, -40.606, 103.88, 145.819, 49.486, -28.433, -175]
  MoveL 454 to (14.54, -76.45, -174.24) mm, rotated rx 42.04 ry 15.1 rz 65.25 deg; joints [-15.499, -40.593, 103.907, 145.8, 49.527, -28.447, -175]
  MoveL 455 to (14.41, -76.1, -174.55) mm, rotated rx 42.04 ry 15.1 rz 65.25 deg; joints [-15.513, -40.594, 103.93, 145.793, 49.548, -28.456, -175]
  MoveL 456 to (14.34, -75.69, -174.82) mm, rotated rx 42.04 ry 15.1 rz 65.25 deg; joints [-15.526, -40.601, 103.96, 145.788, 49.57, -28.467, -175]
  MoveL 457 to (14.36, -74.74, -175.23) mm, rotated rx 42.04 ry 15.1 rz 65.25 deg; joints [-15.548, -40.631, 104.039, 145.785, 49.616, -28.492, -175]
  MoveL 458 to (14.62, -73.58, -175.48) mm, rotated rx 42.04 ry 15.1 rz 65.25 deg; joints [-15.566, -40.682, 104.143, 145.788, 49.665, -28.522, -175]
  MoveL 459 to (15.11, -72.21, -175.56) mm, rotated rx 42.04 ry 15.1 rz 65.25 deg; joints [-15.58, -40.755, 104.273, 145.799, 49.716, -28.558, -175]
  MoveL 460 to (16.5, -68.82, -175.56) mm, rotated rx 42.04 ry 15.1 rz 65.25 deg; joints [-15.605, -40.947, 104.603, 145.834, 49.836, -28.647, -175]
  MoveL 461 to (16.69, -68.4, -175.54) mm, rotated rx 42.04 ry 15.1 rz 65.25 deg; joints [-15.608, -40.972, 104.644, 145.838, 49.85, -28.658, -175]
  MoveL 462 to (16.86, -68.02, -175.52) mm, rotated rx 42.04 ry 15.1 rz 65.25 deg; joints [-15.61, -40.995, 104.681, 145.843, 49.863, -28.668, -175]
  MoveL 463 to (17.05, -67.59, -175.5) mm, rotated rx 42.04 ry 15.1 rz 65.25 deg; joints [-15.612, -41.02, 104.724, 145.848, 49.878, -28.679, -175]
  MoveL 464 to (18.44, -64.2, -175.5) mm, rotated rx 42.04 ry 15.1 rz 65.25 deg; joints [-15.638, -41.212, 105.052, 145.881, 49.997, -28.767, -175]
  MoveL 465 to (18.67, -63.71, -175.48) mm, rotated rx 42.04 ry 15.1 rz 65.25 deg; joints [-15.641, -41.241, 105.101, 145.887, 50.013, -28.779, -175]
  MoveL 466 to (18.92, -63.23, -175.44) mm, rotated rx 42.04 ry 15.1 rz 65.25 deg; joints [-15.644, -41.272, 105.149, 145.892, 50.029, -28.791, -175]
  MoveL 467 to (19.19, -62.82, -175.4) mm, rotated rx 42.04 ry 15.1 rz 65.25 deg; joints [-15.645, -41.302, 105.191, 145.896, 50.04, -28.8, -175]
  MoveL 468 to (19.44, -62.52, -175.33) mm, rotated rx 42.04 ry 15.1 rz 65.25 deg; joints [-15.645, -41.326, 105.224, 145.9, 50.046, -28.806, -175]
  MoveL 469 to (19.58, -62.39, -175.17) mm, rotated rx 42.04 ry 15.1 rz 65.25 deg; joints [-15.64, -41.34, 105.24, 145.908, 50.047, -28.81, -175]
  MoveL 470 to (19.62, -62.4, -174.84) mm, rotated rx 42.04 ry 15.1 rz 65.25 deg; joints [-15.627, -41.344, 105.246, 145.924, 50.046, -28.817, -175]
  MoveL 471 to (19.54, -62.54, -174.33) mm, rotated rx 42.04 ry 15.1 rz 65.25 deg; joints [-15.607, -41.338, 105.241, 145.949, 50.041, -28.828, -175]
  MoveL 472 to (20.36, -62.66, -172.87) mm, rotated rx 42.04 ry 15.1 rz 65.25 deg; joints [-15.551, -41.394, 105.273, 146.005, 50.008, -28.837, -175]
  MoveL 473 to (23.91, -60.28, -172.87) mm, rotated rx 42.04 ry 15.1 rz 65.25 deg; joints [-15.57, -41.68, 105.553, 145.979, 50.008, -28.823, -175]
  MoveL 474 to (25.6, -59.15, -172.82) mm, rotated rx 42.04 ry 15.1 rz 65.25 deg; joints [-15.578, -41.817, 105.687, 145.968, 50.007, -28.817, -175]
  MoveL 475 to (27.25, -58.06, -172.73) mm, rotated rx 42.04 ry 15.1 rz 65.25 deg; joints [-15.583, -41.95, 105.817, 145.96, 50.005, -28.812, -175]
  MoveL 476 to (28.93, -56.94, -172.65) mm, rotated rx 42.04 ry 15.1 rz 65.25 deg; joints [-15.589, -42.086, 105.949, 145.951, 50.004, -28.807, -175]
  MoveL 477 to (30.57, -55.85, -172.55) mm, rotated rx 42.04 ry 15.1 rz 65.25 deg; joints [-15.594, -42.219, 106.079, 145.943, 50.002, -28.802, -175]
  MoveL 478 to (32.32, -54.71, -172.51) mm, rotated rx 42.04 ry 15.1 rz 65.25 deg; joints [-15.602, -42.36, 106.213, 145.931, 49.999, -28.793, -175]
  MoveL 479 to (34.21, -53.57, -172.47) mm, rotated rx 42.04 ry 15.1 rz 65.25 deg; joints [-15.611, -42.509, 106.349, 145.915, 49.99, -28.78, -175]
  MoveL 480 to (36.23, -52.1, -172.31) mm, rotated rx 42.04 ry 15.1 rz 65.25 deg; joints [-15.616, -42.677, 106.519, 145.909, 49.993, -28.779, -175]
  MoveL 481 to (38.1, -50.86, -172.06) mm, rotated rx 42.04 ry 15.1 rz 65.25 deg; joints [-15.617, -42.83, 106.668, 145.906, 49.99, -28.775, -175]
  MoveL 482 to (39.92, -49.64, -171.93) mm, rotated rx 42.04 ry 15.1 rz 65.25 deg; joints [-15.622, -42.978, 106.81, 145.897, 49.986, -28.769, -175]
  MoveL 483 to (41.69, -48.45, -171.69) mm, rotated rx 42.04 ry 15.1 rz 65.25 deg; joints [-15.623, -43.123, 106.951, 145.894, 49.983, -28.765, -175]
  MoveL 484 to (43.46, -47.25, -171.56) mm, rotated rx 42.04 ry 15.1 rz 65.25 deg; joints [-15.628, -43.268, 107.09, 145.886, 49.98, -28.759, -175]
  MoveL 485 to (45.23, -46.06, -171.45) mm, rotated rx 42.04 ry 15.1 rz 65.25 deg; joints [-15.633, -43.412, 107.229, 145.876, 49.976, -28.752, -175]
  MoveL 486 to (46.99, -44.85, -171.21) mm, rotated rx 42.04 ry 15.1 rz 65.25 deg; joints [-15.634, -43.557, 107.37, 145.873, 49.973, -28.748, -175]
  MoveL 487 to (48.75, -43.65, -171.09) mm, rotated rx 42.04 ry 15.1 rz 65.25 deg; joints [-15.639, -43.702, 107.508, 145.864, 49.969, -28.741, -175]
  MoveL 488 to (50.52, -42.45, -170.97) mm, rotated rx 42.04 ry 15.1 rz 65.25 deg; joints [-15.645, -43.846, 107.646, 145.854, 49.965, -28.734, -175]
  MoveL 489 to (52.28, -41.25, -170.85) mm, rotated rx 42.04 ry 15.1 rz 65.25 deg; joints [-15.65, -43.991, 107.784, 145.844, 49.961, -28.726, -175]
  MoveL 490 to (54.03, -40.02, -170.62) mm, rotated rx 42.04 ry 15.1 rz 65.25 deg; joints [-15.652, -44.136, 107.924, 145.841, 49.958, -28.723, -175]
  MoveL 491 to (55.79, -38.81, -170.51) mm, rotated rx 42.04 ry 15.1 rz 65.25 deg; joints [-15.658, -44.28, 108.062, 145.83, 49.953, -28.715, -175]
  MoveL 492 to (57.24, -37.77, -170.26) mm, rotated rx 42.04 ry 15.1 rz 65.25 deg; joints [-15.657, -44.402, 108.182, 145.831, 49.951, -28.714, -175]
  MoveL 493 to (58.57, -36.79, -169.94) mm, rotated rx 42.04 ry 15.1 rz 65.25 deg; joints [-15.652, -44.515, 108.296, 145.836, 49.951, -28.716, -175]
  MoveL 494 to (59.81, -35.83, -169.52) mm, rotated rx 42.04 ry 15.1 rz 65.25 deg; joints [-15.644, -44.624, 108.407, 145.848, 49.951, -28.722, -175]
  MoveL 495 to (58.1, -36.12, -168.56) mm, rotated rx 42.04 ry 15.1 rz 65.25 deg; joints [-15.604, -44.519, 108.369, 145.928, 49.996, -28.79, -175]
  MoveL 496 to (58.65, -35.8, -168.43) mm, rotated rx 42.04 ry 15.1 rz 65.25 deg; joints [-15.601, -44.563, 108.408, 145.928, 49.992, -28.788, -175]
  MoveL 497 to (59.18, -35.57, -168.35) mm, rotated rx 42.04 ry 15.1 rz 65.25 deg; joints [-15.6, -44.603, 108.439, 145.925, 49.984, -28.782, -175]
  MoveL 498 to (59.71, -35.46, -168.31) mm, rotated rx 42.04 ry 15.1 rz 65.25 deg; joints [-15.6, -44.638, 108.458, 145.918, 49.97, -28.77, -175]
  MoveL 499 to (60.24, -35.4, -168.3) mm, rotated rx 42.04 ry 15.1 rz 65.25 deg; joints [-15.6, -44.672, 108.472, 145.909, 49.955, -28.756, -175]
  MoveL 500 to (63.92, -35.37, -168.29) mm, rotated rx 42.04 ry 15.1 rz 65.25 deg; joints [-15.602, -44.891, 108.537, 145.833, 49.826, -28.641, -175]
  MoveL 501 to (64.38, -35.36, -168.28) mm, rotated rx 42.04 ry 15.1 rz 65.25 deg; joints [-15.602, -44.919, 108.545, 145.824, 49.811, -28.627, -175]
  MoveL 502 to (64.8, -35.34, -168.25) mm, rotated rx 42.04 ry 15.1 rz 65.25 deg; joints [-15.601, -44.945, 108.554, 145.817, 49.797, -28.615, -175]
  MoveL 503 to (65.28, -35.34, -168.24) mm, rotated rx 42.04 ry 15.1 rz 65.25 deg; joints [-15.601, -44.974, 108.563, 145.808, 49.78, -28.6, -175]
  MoveL 504 to (65.81, -35.33, -168.24) mm, rotated rx 42.04 ry 15.1 rz 65.25 deg; joints [-15.601, -45.005, 108.572, 145.797, 49.761, -28.584, -175]
  MoveL 505 to (67.38, -35.33, -168.24) mm, rotated rx 42.04 ry 15.1 rz 65.25 deg; joints [-15.602, -45.098, 108.598, 145.764, 49.706, -28.534, -175]
  MoveL 506 to (68.01, -35.32, -168.22) mm, rotated rx 42.04 ry 15.1 rz 65.25 deg; joints [-15.602, -45.136, 108.609, 145.752, 49.684, -28.515, -175]
  MoveL 507 to (68.72, -35.29, -168.18) mm, rotated rx 42.04 ry 15.1 rz 65.25 deg; joints [-15.601, -45.18, 108.624, 145.739, 49.66, -28.494, -175]
  MoveL 508 to (69.37, -35.27, -168.16) mm, rotated rx 42.04 ry 15.1 rz 65.25 deg; joints [-15.6, -45.219, 108.636, 145.727, 49.638, -28.474, -175]
  MoveL 509 to (70.42, -35.27, -168.16) mm, rotated rx 42.04 ry 15.1 rz 65.25 deg; joints [-15.601, -45.281, 108.653, 145.704, 49.601, -28.441, -175]
  MoveL 510 to (71.86, -35.34, -168.24) mm, rotated rx 42.04 ry 15.1 rz 65.25 deg; joints [-15.604, -45.363, 108.669, 145.668, 49.546, -28.389, -175]
  MoveL 511 to (73.03, -35.55, -168.5) mm, rotated rx 42.04 ry 15.1 rz 65.25 deg; joints [-15.613, -45.424, 108.665, 145.626, 49.496, -28.337, -175]
  MoveL 512 to (73.92, -35.9, -168.92) mm, rotated rx 42.04 ry 15.1 rz 65.25 deg; joints [-15.627, -45.462, 108.642, 145.58, 49.449, -28.285, -175]
  MoveL 513 to (74.26, -36.12, -169.19) mm, rotated rx 42.04 ry 15.1 rz 65.25 deg; joints [-15.637, -45.472, 108.623, 145.554, 49.427, -28.259, -175]
  MoveL 514 to (74.53, -36.38, -169.5) mm, rotated rx 42.04 ry 15.1 rz 65.25 deg; joints [-15.647, -45.477, 108.6, 145.528, 49.406, -28.232, -175]
  MoveL 515 to (74.85, -37, -170.26) mm, rotated rx 42.04 ry 15.1 rz 65.25 deg; joints [-15.672, -45.47, 108.538, 145.471, 49.367, -28.179, -175]
  MoveL 516 to (74.9, -37.76, -171.18) mm, rotated rx 42.04 ry 15.1 rz 65.25 deg; joints [-15.702, -45.441, 108.456, 145.409, 49.332, -28.125, -175]
  MoveL 517 to (74.16, -39.7, -173.54) mm, rotated rx 42.04 ry 15.1 rz 65.25 deg; joints [-15.778, -45.315, 108.236, 145.271, 49.273, -28.017, -175]
  MoveL 518 to (72.63, -41.58, -175.89) mm, rotated rx 42.04 ry 15.1 rz 65.25 deg; joints [-15.854, -45.145, 108.006, 145.15, 49.245, -27.935, -175]
  MoveL 519 to (70.63, -42.81, -177.57) mm, rotated rx 42.04 ry 15.1 rz 65.25 deg; joints [-15.908, -44.974, 107.838, 145.085, 49.261, -27.91, -175]
  MoveL 520 to (69.46, -43.18, -178.16) mm, rotated rx 42.04 ry 15.1 rz 65.25 deg; joints [-15.927, -44.888, 107.776, 145.074, 49.286, -27.919, -175]
  MoveL 521 to (68.17, -43.38, -178.58) mm, rotated rx 42.04 ry 15.1 rz 65.25 deg; joints [-15.941, -44.802, 107.73, 145.077, 49.322, -27.942, -175]
  MoveL 522 to (65.26, -43.3, -178.91) mm, rotated rx 42.04 ry 15.1 rz 65.25 deg; joints [-15.953, -44.631, 107.683, 145.123, 49.427, -28.03, -175]
  MoveL 523 to (62.14, -42.9, -178.91) mm, rotated rx 42.04 ry 15.1 rz 65.25 deg; joints [-15.954, -44.461, 107.667, 145.197, 49.554, -28.145, -175]
  MoveL 524 to (61.16, -42.82, -178.96) mm, rotated rx 42.04 ry 15.1 rz 65.25 deg; joints [-15.956, -44.405, 107.656, 145.216, 49.592, -28.178, -175]
  MoveL 525 to (60.64, -42.75, -178.96) mm, rotated rx 42.04 ry 15.1 rz 65.25 deg; joints [-15.957, -44.377, 107.654, 145.228, 49.613, -28.197, -175]
  MoveL 526 to (60.11, -42.69, -178.96) mm, rotated rx 42.04 ry 15.1 rz 65.25 deg; joints [-15.957, -44.347, 107.65, 145.241, 49.634, -28.216, -175]
  MoveL 527 to (59.54, -42.63, -178.99) mm, rotated rx 42.04 ry 15.1 rz 65.25 deg; joints [-15.958, -44.316, 107.646, 145.253, 49.656, -28.236, -175]
  MoveL 528 to (58.9, -42.58, -179.05) mm, rotated rx 42.04 ry 15.1 rz 65.25 deg; joints [-15.96, -44.279, 107.638, 145.264, 49.681, -28.256, -175]
  MoveL 529 to (58.32, -42.53, -179.08) mm, rotated rx 42.04 ry 15.1 rz 65.25 deg; joints [-15.961, -44.246, 107.632, 145.275, 49.703, -28.276, -175]
  MoveL 530 to (57.8, -42.47, -179.09) mm, rotated rx 42.04 ry 15.1 rz 65.25 deg; joints [-15.962, -44.217, 107.628, 145.286, 49.724, -28.294, -175]
  MoveL 531 to (57.32, -42.43, -179.12) mm, rotated rx 42.04 ry 15.1 rz 65.25 deg; joints [-15.963, -44.19, 107.623, 145.296, 49.742, -28.31, -175]
  MoveL 532 to (56.87, -42.41, -179.17) mm, rotated rx 42.04 ry 15.1 rz 65.25 deg; joints [-15.965, -44.163, 107.616, 145.303, 49.759, -28.324, -175]
  MoveL 533 to (56.41, -42.38, -179.21) mm, rotated rx 42.04 ry 15.1 rz 65.25 deg; joints [-15.967, -44.137, 107.61, 145.311, 49.776, -28.338, -175]
  MoveL 534 to (55.9, -42.32, -179.22) mm, rotated rx 42.04 ry 15.1 rz 65.25 deg; joints [-15.967, -44.109, 107.606, 145.322, 49.796, -28.356, -175]
  MoveL 535 to (55.39, -42.27, -179.22) mm, rotated rx 42.04 ry 15.1 rz 65.25 deg; joints [-15.968, -44.08, 107.602, 145.333, 49.816, -28.374, -175]
  MoveL 536 to (54.88, -42.24, -179.23) mm, rotated rx 42.04 ry 15.1 rz 65.25 deg; joints [-15.968, -44.051, 107.595, 145.344, 49.835, -28.391, -175]
  MoveL 537 to (54.39, -42.26, -179.25) mm, rotated rx 42.04 ry 15.1 rz 65.25 deg; joints [-15.968, -44.021, 107.584, 145.353, 49.851, -28.405, -175]
  MoveL 538 to (53.92, -42.34, -179.28) mm, rotated rx 42.04 ry 15.1 rz 65.25 deg; joints [-15.968, -43.991, 107.569, 145.359, 49.863, -28.416, -175]
  MoveL 539 to (53.49, -42.48, -179.33) mm, rotated rx 42.04 ry 15.1 rz 65.25 deg; joints [-15.969, -43.96, 107.548, 145.364, 49.871, -28.423, -175]
  MoveL 540 to (53.06, -42.65, -179.37) mm, rotated rx 42.04 ry 15.1 rz 65.25 deg; joints [-15.969, -43.929, 107.525, 145.367, 49.878, -28.429, -175]
  MoveL 541 to (54.55, -42.33, -180.34) mm, rotated rx 42.04 ry 15.1 rz 65.25 deg; joints [-16.01, -44.02, 107.562, 145.292, 49.844, -28.369, -175]
  MoveL 542 to (53.1, -43.24, -180.72) mm, rotated rx 42.04 ry 15.1 rz 65.25 deg; joints [-16.016, -43.902, 107.45, 145.288, 49.851, -28.371, -175]
  MoveL 543 to (51.53, -44.15, -181) mm, rotated rx 42.04 ry 15.1 rz 65.25 deg; joints [-16.019, -43.777, 107.338, 145.29, 49.862, -28.379, -175]
  MoveL 544 to (49.83, -45.09, -181.2) mm, rotated rx 42.04 ry 15.1 rz 65.25 deg; joints [-16.018, -43.644, 107.223, 145.299, 49.877, -28.392, -175]
  MoveL 545 to (47.94, -46.09, -181.42) mm, rotated rx 42.04 ry 15.1 rz 65.25 deg; joints [-16.018, -43.498, 107.099, 145.31, 49.894, -28.408, -175]
  MoveL 546 to (46.04, -47.06, -181.54) mm, rotated rx 42.04 ry 15.1 rz 65.25 deg; joints [-16.014, -43.354, 106.978, 145.326, 49.913, -28.428, -175]
  MoveL 547 to (44.13, -48.02, -181.65) mm, rotated rx 42.04 ry 15.1 rz 65.25 deg; joints [-16.01, -43.209, 106.857, 145.343, 49.931, -28.448, -175]
  MoveL 548 to (42.23, -49.01, -181.88) mm, rotated rx 42.04 ry 15.1 rz 65.25 deg; joints [-16.01, -43.063, 106.732, 145.353, 49.949, -28.464, -175]
  MoveL 549 to (40.33, -49.97, -182) mm, rotated rx 42.04 ry 15.1 rz 65.25 deg; joints [-16.006, -42.918, 106.611, 145.369, 49.967, -28.483, -175]
  MoveL 550 to (38.42, -50.93, -182.12) mm, rotated rx 42.04 ry 15.1 rz 65.25 deg; joints [-16.002, -42.773, 106.489, 145.385, 49.985, -28.502, -175]
  MoveL 551 to (36.52, -51.9, -182.36) mm, rotated rx 42.04 ry 15.1 rz 65.25 deg; joints [-16.003, -42.628, 106.365, 145.394, 50.002, -28.517, -175]
  MoveL 552 to (34.61, -52.85, -182.48) mm, rotated rx 42.04 ry 15.1 rz 65.25 deg; joints [-15.999, -42.483, 106.243, 145.41, 50.02, -28.536, -175]
  MoveL 553 to (32.7, -53.81, -182.6) mm, rotated rx 42.04 ry 15.1 rz 65.25 deg; joints [-15.995, -42.338, 106.121, 145.425, 50.038, -28.555, -175]
  MoveL 554 to (30.9, -54.7, -182.79) mm, rotated rx 42.04 ry 15.1 rz 65.25 deg; joints [-15.994, -42.201, 106.004, 145.435, 50.055, -28.57, -175]
  MoveL 555 to (29.26, -55.51, -183) mm, rotated rx 42.04 ry 15.1 rz 65.25 deg; joints [-15.995, -42.077, 105.898, 145.443, 50.07, -28.583, -175]
  MoveL 556 to (27.5, -56.38, -183.11) mm, rotated rx 42.04 ry 15.1 rz 65.25 deg; joints [-15.992, -41.944, 105.785, 145.457, 50.086, -28.6, -175]
  MoveL 557 to (25.6, -57.43, -183.11) mm, rotated rx 42.04 ry 15.1 rz 65.25 deg; joints [-15.983, -41.798, 105.655, 145.476, 50.097, -28.616, -175]
  MoveL 558 to (23.15, -58.62, -183.2) mm, rotated rx 42.04 ry 15.1 rz 65.25 deg; joints [-15.975, -41.614, 105.501, 145.498, 50.119, -28.641, -175]
  MoveL 559 to (20.89, -59.6, -183.44) mm, rotated rx 42.04 ry 15.1 rz 65.25 deg; joints [-15.976, -41.447, 105.365, 145.512, 50.145, -28.664, -175]
  MoveL 560 to (19.06, -60.49, -183.62) mm, rotated rx 42.04 ry 15.1 rz 65.25 deg; joints [-15.975, -41.309, 105.247, 145.523, 50.161, -28.679, -175]
  MoveL 561 to (17.37, -61.29, -183.94) mm, rotated rx 42.04 ry 15.1 rz 65.25 deg; joints [-15.98, -41.181, 105.137, 145.525, 50.177, -28.69, -175]
  MoveL 562 to (15.52, -62.17, -184.12) mm, rotated rx 42.04 ry 15.1 rz 65.25 deg; joints [-15.979, -41.042, 105.018, 145.536, 50.194, -28.705, -175]
  MoveL 563 to (13.73, -63, -184.32) mm, rotated rx 42.04 ry 15.1 rz 65.25 deg; joints [-15.979, -40.908, 104.904, 145.545, 50.21, -28.72, -175]
  MoveL 564 to (11.98, -63.79, -184.6) mm, rotated rx 42.04 ry 15.1 rz 65.25 deg; joints [-15.983, -40.777, 104.793, 145.55, 50.228, -28.733, -175]
  MoveL 565 to (11.08, -63.63, -185.37) mm, rotated rx 42.04 ry 15.1 rz 65.25 deg; joints [-16.013, -40.724, 104.775, 145.531, 50.264, -28.745, -175]
  MoveL 566 to (11.29, -63.31, -185.75) mm, rotated rx 42.04 ry 15.1 rz 65.25 deg; joints [-16.03, -40.743, 104.8, 145.513, 50.273, -28.741, -175]
  MoveL 567 to (11.31, -63.23, -185.99) mm, rotated rx 42.04 ry 15.1 rz 65.25 deg; joints [-16.04, -40.745, 104.803, 145.502, 50.276, -28.737, -175]
  MoveL 568 to (11.16, -63.38, -186.12) mm, rotated rx 42.04 ry 15.1 rz 65.25 deg; joints [-16.043, -40.731, 104.785, 145.496, 50.274, -28.732, -175]
  MoveL 569 to (10.85, -63.81, -186.17) mm, rotated rx 42.04 ry 15.1 rz 65.25 deg; joints [-16.042, -40.698, 104.74, 145.492, 50.263, -28.724, -175]
  MoveL 570 to (10.48, -64.36, -186.2) mm, rotated rx 42.04 ry 15.1 rz 65.25 deg; joints [-16.039, -40.658, 104.682, 145.487, 50.248, -28.712, -175]
  MoveL 571 to (9.7, -65.73, -186.2) mm, rotated rx 42.04 ry 15.1 rz 65.25 deg; joints [-16.028, -40.569, 104.545, 145.478, 50.206, -28.683, -175]
  MoveL 572 to (9.42, -66.2, -186.21) mm, rotated rx 42.04 ry 15.1 rz 65.25 deg; joints [-16.024, -40.537, 104.498, 145.474, 50.192, -28.672, -175]
  MoveL 573 to (9.14, -66.66, -186.24) mm, rotated rx 42.04 ry 15.1 rz 65.25 deg; joints [-16.021, -40.506, 104.451, 145.47, 50.179, -28.662, -175]
  MoveL 574 to (8.84, -67.12, -186.29) mm, rotated rx 42.04 ry 15.1 rz 65.25 deg; joints [-16.02, -40.473, 104.403, 145.465, 50.166, -28.652, -175]
  MoveL 575 to (8.52, -67.57, -186.36) mm, rotated rx 42.04 ry 15.1 rz 65.25 deg; joints [-16.019, -40.439, 104.355, 145.46, 50.154, -28.642, -175]
  MoveL 576 to (8.21, -68.03, -186.42) mm, rotated rx 42.04 ry 15.1 rz 65.25 deg; joints [-16.017, -40.405, 104.307, 145.454, 50.141, -28.632, -175]
  MoveL 577 to (7.95, -68.46, -186.44) mm, rotated rx 42.04 ry 15.1 rz 65.25 deg; joints [-16.015, -40.376, 104.263, 145.451, 50.129, -28.622, -175]
  MoveL 578 to (7.72, -68.85, -186.46) mm, rotated rx 42.04 ry 15.1 rz 65.25 deg; joints [-16.012, -40.35, 104.223, 145.447, 50.117, -28.614, -175]
  MoveL 579 to (6.94, -70.21, -186.46) mm, rotated rx 42.04 ry 15.1 rz 65.25 deg; joints [-16.001, -40.26, 104.086, 145.438, 50.075, -28.584, -175]
  MoveL 580 to (6.67, -70.66, -186.47) mm, rotated rx 42.04 ry 15.1 rz 65.25 deg; joints [-15.998, -40.23, 104.04, 145.434, 50.062, -28.574, -175]
  MoveL 581 to (6.42, -71.06, -186.5) mm, rotated rx 42.04 ry 15.1 rz 65.25 deg; joints [-15.996, -40.202, 103.998, 145.43, 50.05, -28.565, -175]
  MoveL 582 to (6.16, -71.43, -186.55) mm, rotated rx 42.04 ry 15.1 rz 65.25 deg; joints [-15.995, -40.174, 103.96, 145.426, 50.04, -28.557, -175]
  MoveL 583 to (5.92, -71.81, -186.59) mm, rotated rx 42.04 ry 15.1 rz 65.25 deg; joints [-15.993, -40.147, 103.92, 145.422, 50.03, -28.548, -175]
  MoveL 584 to (5.66, -72.22, -186.6) mm, rotated rx 42.04 ry 15.1 rz 65.25 deg; joints [-15.991, -40.119, 103.877, 145.419, 50.017, -28.539, -175]
  MoveL 585 to (5.4, -72.68, -186.6) mm, rotated rx 42.04 ry 15.1 rz 65.25 deg; joints [-15.987, -40.089, 103.831, 145.415, 50.003, -28.529, -175]
  MoveL 586 to (3.7, -75.07, -186.94) mm, rotated rx 42.04 ry 15.1 rz 65.25 deg; joints [-15.981, -39.909, 103.576, 145.387, 49.939, -28.476, -175]
  MoveL 587 to (2.76, -75.98, -187.36) mm, rotated rx 42.04 ry 15.1 rz 65.25 deg; joints [-15.989, -39.821, 103.467, 145.367, 49.924, -28.456, -175]
  MoveL 588 to (1.75, -76.71, -187.95) mm, rotated rx 42.04 ry 15.1 rz 65.25 deg; joints [-16.005, -39.733, 103.369, 145.343, 49.92, -28.441, -175]
  MoveL 589 to (-0.46, -77.61, -189.64) mm, rotated rx 42.04 ry 15.1 rz 65.25 deg; joints [-16.06, -39.562, 103.21, 145.282, 49.944, -28.424, -175]
  MoveL 590 to (-2.92, -77.77, -192) mm, rotated rx 42.04 ry 15.1 rz 65.25 deg; joints [-16.146, -39.394, 103.098, 145.206, 50.011, -28.424, -175]
  MoveL 591 to (-4.94, -77.27, -194.36) mm, rotated rx 42.04 ry 15.1 rz 65.25 deg; joints [-16.237, -39.274, 103.054, 145.133, 50.097, -28.438, -175]
  MoveL 592 to (-5.53, -76.8, -195.29) mm, rotated rx 42.04 ry 15.1 rz 65.25 deg; joints [-16.275, -39.247, 103.066, 145.105, 50.138, -28.449, -175]
  MoveL 593 to (-5.84, -76.19, -196.05) mm, rotated rx 42.04 ry 15.1 rz 65.25 deg; joints [-16.308, -39.243, 103.099, 145.084, 50.177, -28.461, -175]
  MoveL 594 to (-5.89, -75.83, -196.37) mm, rotated rx 42.04 ry 15.1 rz 65.25 deg; joints [-16.323, -39.249, 103.124, 145.075, 50.197, -28.469, -175]
  MoveL 595 to (-5.87, -75.43, -196.64) mm, rotated rx 42.04 ry 15.1 rz 65.25 deg; joints [-16.336, -39.261, 103.155, 145.068, 50.215, -28.476, -175]
  MoveL 596 to (-5.62, -74.52, -197.06) mm, rotated rx 42.04 ry 15.1 rz 65.25 deg; joints [-16.359, -39.302, 103.233, 145.059, 50.252, -28.493, -175]
  MoveL 597 to (-5.08, -73.48, -197.32) mm, rotated rx 42.04 ry 15.1 rz 65.25 deg; joints [-16.377, -39.365, 103.334, 145.055, 50.287, -28.513, -175]
  MoveL 598 to (-4.26, -72.28, -197.4) mm, rotated rx 42.04 ry 15.1 rz 65.25 deg; joints [-16.39, -39.451, 103.456, 145.057, 50.32, -28.534, -175]
  MoveL 599 to (-3.32, -71.03, -197.4) mm, rotated rx 42.04 ry 15.1 rz 65.25 deg; joints [-16.401, -39.547, 103.588, 145.062, 50.353, -28.556, -175]
  MoveL 600 to (-3, -70.61, -197.4) mm, rotated rx 42.04 ry 15.1 rz 65.25 deg; joints [-16.404, -39.579, 103.633, 145.063, 50.363, -28.564, -175]
  MoveL 601 to (-2.63, -70.17, -197.36) mm, rotated rx 42.04 ry 15.1 rz 65.25 deg; joints [-16.406, -39.615, 103.681, 145.066, 50.374, -28.571, -175]
  MoveL 602 to (-2.2, -69.68, -197.3) mm, rotated rx 42.04 ry 15.1 rz 65.25 deg; joints [-16.408, -39.656, 103.734, 145.07, 50.384, -28.58, -175]
  MoveL 603 to (-1.85, -69.24, -197.27) mm, rotated rx 42.04 ry 15.1 rz 65.25 deg; joints [-16.411, -39.691, 103.782, 145.072, 50.395, -28.587, -175]
  MoveL 604 to (-1.52, -68.82, -197.27) mm, rotated rx 42.04 ry 15.1 rz 65.25 deg; joints [-16.414, -39.724, 103.826, 145.074, 50.406, -28.595, -175]
  MoveL 605 to (-1.21, -68.41, -197.26) mm, rotated rx 42.04 ry 15.1 rz 65.25 deg; joints [-16.417, -39.756, 103.869, 145.076, 50.416, -28.602, -175]
  MoveL 606 to (-0.87, -68.03, -197.21) mm, rotated rx 42.04 ry 15.1 rz 65.25 deg; joints [-16.419, -39.788, 103.912, 145.079, 50.424, -28.609, -175]
  MoveL 607 to (-0.53, -67.66, -197.13) mm, rotated rx 42.04 ry 15.1 rz 65.25 deg; joints [-16.419, -39.821, 103.953, 145.083, 50.432, -28.615, -175]
  MoveL 608 to (-0.18, -67.3, -197.04) mm, rotated rx 42.04 ry 15.1 rz 65.25 deg; joints [-16.418, -39.854, 103.995, 145.087, 50.438, -28.622, -175]
  MoveL 609 to (0.17, -66.92, -196.97) mm, rotated rx 42.04 ry 15.1 rz 65.25 deg; joints [-16.419, -39.887, 104.037, 145.091, 50.446, -28.628, -175]
  MoveL 610 to (0.51, -66.51, -196.94) mm, rotated rx 42.04 ry 15.1 rz 65.25 deg; joints [-16.421, -39.92, 104.081, 145.094, 50.456, -28.635, -175]
  MoveL 611 to (0.83, -66.1, -196.92) mm, rotated rx 42.04 ry 15.1 rz 65.25 deg; joints [-16.424, -39.952, 104.125, 145.096, 50.466, -28.642, -175]
  MoveL 612 to (2.4, -64.09, -196.92) mm, rotated rx 42.04 ry 15.1 rz 65.25 deg; joints [-16.441, -40.109, 104.337, 145.102, 50.515, -28.676, -175]
  MoveL 613 to (2.68, -63.82, -196.89) mm, rotated rx 42.04 ry 15.1 rz 65.25 deg; joints [-16.442, -40.134, 104.367, 145.102, 50.519, -28.679, -175]
  MoveL 614 to (2.82, -63.72, -196.78) mm, rotated rx 42.04 ry 15.1 rz 65.25 deg; joints [-16.439, -40.146, 104.38, 145.107, 50.52, -28.681, -175]
  MoveL 615 to (2.76, -63.79, -196.55) mm, rotated rx 42.04 ry 15.1 rz 65.25 deg; joints [-16.429, -40.143, 104.378, 145.119, 50.519, -28.687, -175]
  MoveL 616 to (2.47, -64.01, -196.19) mm, rotated rx 42.04 ry 15.1 rz 65.25 deg; joints [-16.414, -40.122, 104.359, 145.139, 50.517, -28.696, -175]
  MoveL 617 to (3.22, -64.19, -195.45) mm, rotated rx 42.04 ry 15.1 rz 65.25 deg; joints [-16.385, -40.165, 104.373, 145.159, 50.485, -28.686, -175]
  MoveL 618 to (5.22, -63.5, -195.43) mm, rotated rx 42.04 ry 15.1 rz 65.25 deg; joints [-16.391, -40.306, 104.477, 145.134, 50.456, -28.656, -175]
  MoveL 619 to (7.3, -62.82, -195.3) mm, rotated rx 42.04 ry 15.1 rz 65.25 deg; joints [-16.393, -40.452, 104.583, 145.114, 50.424, -28.627, -175]
  MoveL 620 to (9.47, -62.15, -195.04) mm, rotated rx 42.04 ry 15.1 rz 65.25 deg; joints [-16.389, -40.604, 104.693, 145.098, 50.389, -28.597, -175]
  MoveL 621 to (11.48, -61.49, -194.91) mm, rotated rx 42.04 ry 15.1 rz 65.25 deg; joints [-16.391, -40.745, 104.796, 145.078, 50.358, -28.568, -175]
  MoveL 622 to (13.43, -60.86, -194.65) mm, rotated rx 42.04 ry 15.1 rz 65.25 deg; joints [-16.387, -40.882, 104.896, 145.065, 50.327, -28.542, -175]
  MoveL 623 to (15.44, -60.23, -194.29) mm, rotated rx 42.04 ry 15.1 rz 65.25 deg; joints [-16.38, -41.024, 105, 145.056, 50.294, -28.518, -175]
  MoveL 624 to (17.47, -59.54, -194.15) mm, rotated rx 42.04 ry 15.1 rz 65.25 deg; joints [-16.381, -41.167, 105.104, 145.036, 50.262, -28.488, -175]
  MoveL 625 to (19.48, -58.86, -194.05) mm, rotated rx 42.04 ry 15.1 rz 65.25 deg; joints [-16.384, -41.308, 105.207, 145.014, 50.231, -28.458, -175]
  MoveL 626 to (21.51, -58.17, -193.9) mm, rotated rx 42.04 ry 15.1 rz 65.25 deg; joints [-16.385, -41.451, 105.311, 144.994, 50.2, -28.428, -175]
  MoveL 627 to (23.5, -57.52, -193.62) mm, rotated rx 42.04 ry 15.1 rz 65.25 deg; joints [-16.38, -41.592, 105.413, 144.981, 50.167, -28.401, -175]
  MoveL 628 to (25.55, -56.78, -193.28) mm, rotated rx 42.04 ry 15.1 rz 65.25 deg; joints [-16.374, -41.74, 105.525, 144.971, 50.136, -28.378, -175]
  MoveL 629 to (27.55, -56.07, -193.1) mm, rotated rx 42.04 ry 15.1 rz 65.25 deg; joints [-16.374, -41.882, 105.63, 144.953, 50.105, -28.349, -175]
  MoveL 630 to (29.58, -55.37, -192.99) mm, rotated rx 42.04 ry 15.1 rz 65.25 deg; joints [-16.377, -42.025, 105.733, 144.931, 50.073, -28.318, -175]
  MoveL 631 to (31.58, -54.67, -192.91) mm, rotated rx 42.04 ry 15.1 rz 65.25 deg; joints [-16.381, -42.167, 105.834, 144.907, 50.042, -28.286, -175]
  MoveL 632 to (33.6, -53.94, -192.69) mm, rotated rx 42.04 ry 15.1 rz 65.25 deg; joints [-16.379, -42.311, 105.941, 144.89, 50.01, -28.258, -175]
  MoveL 633 to (35.6, -53.23, -192.56) mm, rotated rx 42.04 ry 15.1 rz 65.25 deg; joints [-16.381, -42.453, 106.043, 144.869, 49.978, -28.228, -175]
  MoveL 634 to (37.62, -52.52, -192.48) mm, rotated rx 42.04 ry 15.1 rz 65.25 deg; joints [-16.385, -42.596, 106.145, 144.845, 49.946, -28.195, -175]
  MoveL 635 to (39.61, -51.78, -192.25) mm, rotated rx 42.04 ry 15.1 rz 65.25 deg; joints [-16.383, -42.739, 106.251, 144.828, 49.915, -28.168, -175]
  MoveL 636 to (41.63, -51.03, -192.02) mm, rotated rx 42.04 ry 15.1 rz 65.25 deg; joints [-16.382, -42.885, 106.359, 144.812, 49.883, -28.14, -175]
  MoveL 637 to (43.68, -50.28, -191.87) mm, rotated rx 42.04 ry 15.1 rz 65.25 deg; joints [-16.383, -43.031, 106.464, 144.791, 49.85, -28.109, -175]
  MoveL 638 to (45.43, -49.61, -191.74) mm, rotated rx 42.04 ry 15.1 rz 65.25 deg; joints [-16.385, -43.157, 106.557, 144.772, 49.824, -28.083, -175]
  MoveL 639 to (46.94, -48.96, -191.53) mm, rotated rx 42.04 ry 15.1 rz 65.25 deg; joints [-16.383, -43.269, 106.645, 144.763, 49.803, -28.066, -175]
  MoveL 640 to (48.23, -48.33, -191.21) mm, rotated rx 42.04 ry 15.1 rz 65.25 deg; joints [-16.376, -43.368, 106.729, 144.764, 49.79, -28.058, -175]
  MoveL 641 to (46.78, -48.59, -190.25) mm, rotated rx 42.04 ry 15.1 rz 65.25 deg; joints [-16.337, -43.281, 106.698, 144.838, 49.825, -28.118, -175]
  MoveL 642 to (47.25, -48.43, -190.25) mm, rotated rx 42.04 ry 15.1 rz 65.25 deg; joints [-16.338, -43.314, 106.72, 144.831, 49.817, -28.11, -175]
  MoveL 643 to (47.73, -48.31, -190.25) mm, rotated rx 42.04 ry 15.1 rz 65.25 deg; joints [-16.339, -43.347, 106.74, 144.824, 49.806, -28.1, -175]
  MoveL 644 to (48.26, -48.27, -190.22) mm, rotated rx 42.04 ry 15.1 rz 65.25 deg; joints [-16.339, -43.379, 106.753, 144.815, 49.79, -28.085, -175]
  MoveL 645 to (48.82, -48.29, -190.18) mm, rotated rx 42.04 ry 15.1 rz 65.25 deg; joints [-16.337, -43.412, 106.762, 144.805, 49.77, -28.068, -175]
  MoveL 646 to (49.43, -48.37, -190.13) mm, rotated rx 42.04 ry 15.1 rz 65.25 deg; joints [-16.335, -43.446, 106.767, 144.794, 49.746, -28.047, -175]
  MoveL 647 to (50, -48.49, -190.09) mm, rotated rx 42.04 ry 15.1 rz 65.25 deg; joints [-16.333, -43.476, 106.767, 144.782, 49.722, -28.026, -175]
  MoveL 648 to (50.54, -48.62, -190.07) mm, rotated rx 42.04 ry 15.1 rz 65.25 deg; joints [-16.332, -43.504, 106.766, 144.769, 49.697, -28.004, -175]
  MoveL 649 to (51.05, -48.75, -190.07) mm, rotated rx 42.04 ry 15.1 rz 65.25 deg; joints [-16.331, -43.529, 106.763, 144.756, 49.674, -27.983, -175]
  MoveL 650 to (51.56, -48.89, -190.07) mm, rotated rx 42.04 ry 15.1 rz 65.25 deg; joints [-16.33, -43.555, 106.761, 144.743, 49.651, -27.962, -175]
  MoveL 651 to (52.14, -49, -190.02) mm, rotated rx 42.04 ry 15.1 rz 65.25 deg; joints [-16.328, -43.585, 106.761, 144.731, 49.626, -27.941, -175]
  MoveL 652 to (52.79, -49.11, -189.94) mm, rotated rx 42.04 ry 15.1 rz 65.25 deg; joints [-16.324, -43.621, 106.765, 144.72, 49.599, -27.919, -175]
  MoveL 653 to (53.3, -49.21, -189.89) mm, rotated rx 42.04 ry 15.1 rz 65.25 deg; joints [-16.322, -43.648, 106.766, 144.71, 49.577, -27.9, -175]
  MoveL 654 to (53.71, -49.3, -189.86) mm, rotated rx 42.04 ry 15.1 rz 65.25 deg; joints [-16.32, -43.669, 106.765, 144.701, 49.559, -27.884, -175]
  MoveL 655 to (54.18, -49.42, -189.85) mm, rotated rx 42.04 ry 15.1 rz 65.25 deg; joints [-16.319, -43.693, 106.763, 144.69, 49.537, -27.865, -175]
  MoveL 656 to (54.68, -49.55, -189.85) mm, rotated rx 42.04 ry 15.1 rz 65.25 deg; joints [-16.318, -43.718, 106.761, 144.677, 49.514, -27.844, -175]
